SPLINE
SPL {X  -129.118, Y  +765.975, Z    +0.000, E1   +43.713, E3 -248326.138}
SPL {X  -146.252, Y  +736.362, Z    +0.000, E1   +34.795, E3 -248375.316}
SPL {X  -154.088, Y  +714.555, Z    +0.000, E1   +26.177, E3 -248389.332}
SPL {X  -156.688, Y  +703.837, Z    +0.000, E1   +21.096, E3 -248393.504}
SPL {X  -159.039, Y  +688.920, Z    +0.000, E1   +13.016, E3 -248397.436}
SPL {X  -159.888, Y  +677.224, Z    +0.000, E1    +5.773, E3 -248399.149}
SPL {X  -159.990, Y  +671.755, Z    +0.000, E1    +1.905, E3 -248399.552}
SPL {X  -159.990, Y  +669.598, Z    +0.000, E1    +0.205, E3 -248399.625}
SPL {X  -159.990, Y  +667.097, Z    +0.000, E1    -2.190, E3 -248399.720}
SPL {X  -159.990, Y  +662.904, Z    +0.000, E1    -7.618, E3 -248400.008}
SPL {X  -159.990, Y  +658.509, Z    +0.000, E1   -13.882, E3 -248400.544}
SPL {X  -159.990, Y  +652.317, Z    +0.000, E1   -22.778, E3 -248401.679}
SPL {X  -159.990, Y  +640.689, Z    +0.000, E1   -37.390, E3 -248403.222}
SPL {X  -159.990, Y  +585.634, Z    +0.000, E1   -68.681, E3 -248403.846}
SPL {X  -159.990, Y  +457.771, Z    +0.000, E1   -68.079, E3 -248494.407}
SPL {X  -159.990, Y  +453.218, Z    +0.000, E1   -67.322, E3 -248504.843}
SPL {X  -159.990, Y  +450.256, Z    +0.000, E1   -66.188, E3 -248516.775}
SPL {X  -159.990, Y  +445.667, Z    +0.000, E1   -65.356, E3 -248527.687}
SPL {X  -159.990, Y  +439.738, Z    +0.000, E1   -64.716, E3 -248538.500}
SPL {X  -159.990, Y  +435.528, Z    +0.000, E1   -63.972, E3 -248548.376}
SPL {X  -159.990, Y  +429.021, Z    +0.000, E1   -63.228, E3 -248560.989}
SPL {X  -159.990, Y  +423.267, Z    +0.000, E1   -62.365, E3 -248573.287}
SPL {X  -159.990, Y  +418.218, Z    +0.000, E1   -61.769, E3 -248583.299}
SPL {X  -159.990, Y  +412.274, Z    +0.000, E1   -61.123, E3 -248594.703}
SPL {X  -159.990, Y  +408.631, Z    +0.000, E1   -60.233, E3 -248605.165}
SPL {X  -159.990, Y  +404.834, Z    +0.000, E1   -59.529, E3 -248614.620}
SPL {X  -159.990, Y  +397.866, Z    +0.000, E1   -58.924, E3 -248627.708}
SPL {X  -159.990, Y  +387.403, Z    +0.000, E1   -58.805, E3 -248641.803}
SPL {X  -159.948, Y  +378.844, Z    +0.000, E1   -58.798, E3 -248652.843}
SPL {X  -159.570, Y  +370.916, Z    +0.000, E1   -58.738, E3 -248663.438}
SPL {X  -158.865, Y  +363.563, Z    +0.000, E1   -58.615, E3 -248673.648}
SPL {X  -157.976, Y  +357.197, Z    +0.000, E1   -58.476, E3 -248682.748}
SPL {X  -156.730, Y  +350.368, Z    +0.000, E1   -58.276, E3 -248692.844}
SPL {X  -155.026, Y  +342.956, Z    +0.000, E1   -58.003, E3 -248704.116}
SPL {X  -152.946, Y  +335.551, Z    +0.000, E1   -57.653, E3 -248715.764}
SPL {X  -150.899, Y  +329.336, Z    +0.000, E1   -57.290, E3 -248725.829}
SPL {X  -149.179, Y  +324.687, Z    +0.000, E1   -56.983, E3 -248733.519}
SPL {X  -147.281, Y  +320.009, Z    +0.000, E1   -56.662, E3 -248741.345}
SPL {X  -144.114, Y  +313.017, Z    +0.000, E1   -56.131, E3 -248753.312}
SPL {X  -140.858, Y  +306.633, Z    +0.000, E1   -55.477, E3 -248764.608}
SPL {X  -138.338, Y  +302.130, Z    +0.000, E1   -54.992, E3 -248772.657}
SPL {X  -124.427, Y  +281.929, Z    +0.000, E1   -46.852, E3 -248876.894}
ENDSPLINE

SPLINE
SPL {X  -148.251, Y  +322.346, Z    +0.000, E1   -33.039, E3 -248964.819}
SPL {X  -157.534, Y  +354.574, Z    +0.000, E1   -18.815, E3 -248981.648}
SPL {X  -159.548, Y  +370.614, Z    +0.000, E1    -9.656, E3 -248985.273}
SPL {X  -159.973, Y  +380.173, Z    +0.000, E1    -3.469, E3 -248986.340}
SPL {X  -159.990, Y  +384.791, Z    +0.000, E1    +0.055, E3 -248986.559}
SPL {X  -159.990, Y  +388.179, Z    +0.000, E1    +3.660, E3 -248986.719}
SPL {X  -159.990, Y  +394.222, Z    +0.000, E1   +11.674, E3 -248987.313}
SPL {X  -159.990, Y  +403.976, Z    +0.000, E1   +25.456, E3 -248989.192}
SPL {X  -159.990, Y  +417.120, Z    +0.000, E1   +39.678, E3 -248993.224}
SPL {X  -159.990, Y  +456.927, Z    +0.000, E1   +55.382, E3 -249015.084}
SPL {X  -159.990, Y  +530.047, Z    +0.000, E1   +58.901, E3 -249084.918}
SPL {X  -159.990, Y  +538.035, Z    +0.000, E1   +58.900, E3 -249095.143}
SPL {X  -159.990, Y  +546.883, Z    +0.000, E1   +58.912, E3 -249106.447}
SPL {X  -159.990, Y  +555.949, Z    +0.000, E1   +58.900, E3 -249118.066}
SPL {X  -159.990, Y  +563.718, Z    +0.000, E1   +58.903, E3 -249127.986}
SPL {X  -159.990, Y  +571.529, Z    +0.000, E1   +58.906, E3 -249137.970}
SPL {X  -159.990, Y  +579.859, Z    +0.000, E1   +58.907, E3 -249148.630}
SPL {X  -159.990, Y  +588.526, Z    +0.000, E1   +58.910, E3 -249159.703}
SPL {X  -159.990, Y  +596.521, Z    +0.000, E1   +58.902, E3 -249169.962}
SPL {X  -159.990, Y  +605.444, Z    +0.000, E1   +58.918, E3 -249181.352}
SPL {X  -159.990, Y  +613.908, Z    +0.000, E1   +58.900, E3 -249192.211}
SPL {X  -159.990, Y  +621.342, Z    +0.000, E1   +58.904, E3 -249201.719}
SPL {X  -159.990, Y  +629.920, Z    +0.000, E1   +58.912, E3 -249212.692}
SPL {X  -159.990, Y  +642.398, Z    +0.000, E1   +58.947, E3 -249228.599}
SPL {X  -159.990, Y  +654.206, Z    +0.000, E1   +58.908, E3 -249243.770}
SPL {X  -159.990, Y  +661.562, Z    +0.000, E1   +58.900, E3 -249253.199}
SPL {X  -159.990, Y  +670.328, Z    +0.000, E1   +58.911, E3 -249264.398}
SPL {X  -159.795, Y  +679.404, Z    +0.000, E1   +58.876, E3 -249276.223}
SPL {X  -159.282, Y  +686.534, Z    +0.000, E1   +58.787, E3 -249285.897}
SPL {X  -158.463, Y  +693.553, Z    +0.000, E1   +58.665, E3 -249295.738}
SPL {X  -157.294, Y  +700.745, Z    +0.000, E1   +58.469, E3 -249306.188}
SPL {X  -156.031, Y  +706.871, Z    +0.000, E1   +58.260, E3 -249315.334}
SPL {X  -154.558, Y  +712.835, Z    +0.000, E1   +58.028, E3 -249324.461}
SPL {X  -152.750, Y  +719.085, Z    +0.000, E1   +57.721, E3 -249334.307}
SPL {X  -150.741, Y  +725.111, Z    +0.000, E1   +57.387, E3 -249344.011}
SPL {X  -148.665, Y  +730.623, Z    +0.000, E1   +57.007, E3 -249353.160}
SPL {X  -146.664, Y  +735.425, Z    +0.000, E1   +56.657, E3 -249361.250}
SPL {X  -143.496, Y  +742.251, Z    +0.000, E1   +56.124, E3 -249372.943}
SPL {X  -140.752, Y  +747.564, Z    +0.000, E1   +55.554, E3 -249382.350}
SPL {X  -138.492, Y  +751.605, Z    +0.000, E1   +55.137, E3 -249389.541}
SPL {X  -124.324, Y  +772.199, Z    +0.000, E1   +48.708, E3 -249468.549}
ENDSPLINE

SPLINE
SPL {X  -129.118, Y  +765.975, Z    +0.000, E1   +43.713, E3 -249533.035}
SPL {X  -146.252, Y  +736.362, Z    +0.000, E1   +34.795, E3 -249582.213}
SPL {X  -155.916, Y  +707.374, Z    +0.000, E1   +22.878, E3 -249599.098}
SPL {X  -159.039, Y  +688.920, Z    +0.000, E1   +13.016, E3 -249604.333}
SPL {X  -159.888, Y  +677.224, Z    +0.000, E1    +5.773, E3 -249606.045}
SPL {X  -159.990, Y  +670.275, Z    +0.000, E1    +0.854, E3 -249606.499}
SPL {X  -159.990, Y  +667.097, Z    +0.000, E1    -2.190, E3 -249606.617}
SPL {X  -159.990, Y  +662.904, Z    +0.000, E1    -7.618, E3 -249606.905}
SPL {X  -159.990, Y  +658.509, Z    +0.000, E1   -13.882, E3 -249607.441}
SPL {X  -159.990, Y  +652.317, Z    +0.000, E1   -22.778, E3 -249608.576}
SPL {X  -159.990, Y  +640.689, Z    +0.000, E1   -37.390, E3 -249610.119}
SPL {X  -159.990, Y  +585.634, Z    +0.000, E1   -68.681, E3 -249610.743}
SPL {X  -159.990, Y  +457.771, Z    +0.000, E1   -68.079, E3 -249701.304}
SPL {X  -159.990, Y  +453.218, Z    +0.000, E1   -67.322, E3 -249711.739}
SPL {X  -159.990, Y  +450.256, Z    +0.000, E1   -66.188, E3 -249723.672}
SPL {X  -159.990, Y  +445.667, Z    +0.000, E1   -65.356, E3 -249734.584}
SPL {X  -159.990, Y  +439.738, Z    +0.000, E1   -64.716, E3 -249745.397}
SPL {X  -159.990, Y  +435.528, Z    +0.000, E1   -63.972, E3 -249755.272}
SPL {X  -159.990, Y  +429.021, Z    +0.000, E1   -63.228, E3 -249767.885}
SPL {X  -159.990, Y  +423.267, Z    +0.000, E1   -62.365, E3 -249780.183}
SPL {X  -159.990, Y  +418.218, Z    +0.000, E1   -61.769, E3 -249790.196}
SPL {X  -159.990, Y  +412.274, Z    +0.000, E1   -61.123, E3 -249801.600}
SPL {X  -159.990, Y  +408.631, Z    +0.000, E1   -60.233, E3 -249812.062}
SPL {X  -159.990, Y  +404.834, Z    +0.000, E1   -59.529, E3 -249821.517}
SPL {X  -159.990, Y  +397.866, Z    +0.000, E1   -58.924, E3 -249834.604}
SPL {X  -159.990, Y  +387.403, Z    +0.000, E1   -58.805, E3 -249848.700}
SPL {X  -159.948, Y  +378.844, Z    +0.000, E1   -58.798, E3 -249859.739}
SPL {X  -159.570, Y  +370.916, Z    +0.000, E1   -58.738, E3 -249870.335}
SPL {X  -158.865, Y  +363.563, Z    +0.000, E1   -58.615, E3 -249880.544}
SPL {X  -157.976, Y  +357.197, Z    +0.000, E1   -58.476, E3 -249889.645}
SPL {X  -156.730, Y  +350.368, Z    +0.000, E1   -58.276, E3 -249899.740}
SPL {X  -155.026, Y  +342.956, Z    +0.000, E1   -58.003, E3 -249911.012}
SPL {X  -152.946, Y  +335.551, Z    +0.000, E1   -57.653, E3 -249922.660}
SPL {X  -150.899, Y  +329.336, Z    +0.000, E1   -57.290, E3 -249932.726}
SPL {X  -149.179, Y  +324.687, Z    +0.000, E1   -56.983, E3 -249940.415}
SPL {X  -147.281, Y  +320.009, Z    +0.000, E1   -56.662, E3 -249948.241}
SPL {X  -144.114, Y  +313.017, Z    +0.000, E1   -56.131, E3 -249960.209}
SPL {X  -140.858, Y  +306.633, Z    +0.000, E1   -55.477, E3 -249971.504}
SPL {X  -138.338, Y  +302.130, Z    +0.000, E1   -54.992, E3 -249979.554}
SPL {X  -124.427, Y  +281.929, Z    +0.000, E1   -46.852, E3 -250083.790}
ENDSPLINE

SPLINE
SPL {X  -148.251, Y  +322.346, Z    +0.000, E1   -33.039, E3 -250171.715}
SPL {X  -156.481, Y  +349.177, Z    +0.000, E1   -21.514, E3 -250186.898}
SPL {X  -159.327, Y  +367.953, Z    +0.000, E1   -11.342, E3 -250191.690}
SPL {X  -159.973, Y  +380.173, Z    +0.000, E1    -3.469, E3 -250193.237}
SPL {X  -159.990, Y  +384.078, Z    +0.000, E1    -0.490, E3 -250193.434}
SPL {X  -159.990, Y  +386.348, Z    +0.000, E1    +1.571, E3 -250193.515}
SPL {X  -159.990, Y  +391.422, Z    +0.000, E1    +7.757, E3 -250193.889}
SPL {X  -159.990, Y  +399.099, Z    +0.000, E1   +18.787, E3 -250194.996}
SPL {X  -159.990, Y  +406.316, Z    +0.000, E1   +28.569, E3 -250196.673}
SPL {X  -159.990, Y  +417.120, Z    +0.000, E1   +39.678, E3 -250200.120}
SPL {X  -159.990, Y  +456.927, Z    +0.000, E1   +55.382, E3 -250221.980}
SPL {X  -159.990, Y  +530.047, Z    +0.000, E1   +58.901, E3 -250291.814}
SPL {X  -159.990, Y  +538.035, Z    +0.000, E1   +58.900, E3 -250302.040}
SPL {X  -159.990, Y  +546.883, Z    +0.000, E1   +58.912, E3 -250313.343}
SPL {X  -159.990, Y  +555.949, Z    +0.000, E1   +58.900, E3 -250324.963}
SPL {X  -159.990, Y  +563.718, Z    +0.000, E1   +58.903, E3 -250334.883}
SPL {X  -159.990, Y  +571.529, Z    +0.000, E1   +58.906, E3 -250344.867}
SPL {X  -159.990, Y  +579.859, Z    +0.000, E1   +58.907, E3 -250355.526}
SPL {X  -159.990, Y  +588.526, Z    +0.000, E1   +58.910, E3 -250366.600}
SPL {X  -159.990, Y  +596.521, Z    +0.000, E1   +58.902, E3 -250376.859}
SPL {X  -159.990, Y  +605.444, Z    +0.000, E1   +58.918, E3 -250388.248}
SPL {X  -159.990, Y  +613.908, Z    +0.000, E1   +58.900, E3 -250399.108}
SPL {X  -159.990, Y  +621.342, Z    +0.000, E1   +58.904, E3 -250408.616}
SPL {X  -159.990, Y  +629.920, Z    +0.000, E1   +58.912, E3 -250419.588}
SPL {X  -159.990, Y  +638.424, Z    +0.000, E1   +58.901, E3 -250430.488}
SPL {X  -159.990, Y  +645.995, Z    +0.000, E1   +58.900, E3 -250440.176}
SPL {X  -159.990, Y  +654.206, Z    +0.000, E1   +58.908, E3 -250450.667}
SPL {X  -159.990, Y  +661.562, Z    +0.000, E1   +58.900, E3 -250460.095}
SPL {X  -159.990, Y  +670.328, Z    +0.000, E1   +58.911, E3 -250471.294}
SPL {X  -159.795, Y  +679.404, Z    +0.000, E1   +58.876, E3 -250483.119}
SPL {X  -159.282, Y  +686.534, Z    +0.000, E1   +58.787, E3 -250492.793}
SPL {X  -158.463, Y  +693.553, Z    +0.000, E1   +58.665, E3 -250502.634}
SPL {X  -157.294, Y  +700.745, Z    +0.000, E1   +58.469, E3 -250513.084}
SPL {X  -156.031, Y  +706.871, Z    +0.000, E1   +58.260, E3 -250522.230}
SPL {X  -154.558, Y  +712.835, Z    +0.000, E1   +58.028, E3 -250531.357}
SPL {X  -152.750, Y  +719.085, Z    +0.000, E1   +57.721, E3 -250541.203}
SPL {X  -150.741, Y  +725.111, Z    +0.000, E1   +57.387, E3 -250550.907}
SPL {X  -148.665, Y  +730.623, Z    +0.000, E1   +57.007, E3 -250560.056}
SPL {X  -146.664, Y  +735.425, Z    +0.000, E1   +56.657, E3 -250568.146}
SPL {X  -143.496, Y  +742.251, Z    +0.000, E1   +56.124, E3 -250579.839}
SPL {X  -140.752, Y  +747.564, Z    +0.000, E1   +55.554, E3 -250589.247}
SPL {X  -138.492, Y  +751.605, Z    +0.000, E1   +55.137, E3 -250596.438}
SPL {X  -124.324, Y  +772.199, Z    +0.000, E1   +48.708, E3 -250675.446}
ENDSPLINE

SPLINE
SPL {X  -129.118, Y  +765.975, Z    +0.000, E1   +43.713, E3 -250739.931}
SPL {X  -146.252, Y  +736.362, Z    +0.000, E1   +34.795, E3 -250789.109}
SPL {X  -154.088, Y  +714.555, Z    +0.000, E1   +26.177, E3 -250803.125}
SPL {X  -156.688, Y  +703.837, Z    +0.000, E1   +21.096, E3 -250807.297}
SPL {X  -159.039, Y  +688.920, Z    +0.000, E1   +13.016, E3 -250811.229}
SPL {X  -159.888, Y  +677.224, Z    +0.000, E1    +5.773, E3 -250812.942}
SPL {X  -159.990, Y  +671.755, Z    +0.000, E1    +1.905, E3 -250813.345}
SPL {X  -159.990, Y  +668.898, Z    +0.000, E1    -0.346, E3 -250813.439}
SPL {X  -159.990, Y  +666.084, Z    +0.000, E1    -3.512, E3 -250813.562}
SPL {X  -159.990, Y  +662.904, Z    +0.000, E1    -7.618, E3 -250813.801}
SPL {X  -159.990, Y  +658.509, Z    +0.000, E1   -13.882, E3 -250814.337}
SPL {X  -159.990, Y  +652.317, Z    +0.000, E1   -22.778, E3 -250815.473}
SPL {X  -159.990, Y  +640.689, Z    +0.000, E1   -37.390, E3 -250817.015}
SPL {X  -159.990, Y  +585.634, Z    +0.000, E1   -68.681, E3 -250817.639}
SPL {X  -159.990, Y  +457.771, Z    +0.000, E1   -68.079, E3 -250908.201}
SPL {X  -159.990, Y  +453.218, Z    +0.000, E1   -67.322, E3 -250918.636}
SPL {X  -159.990, Y  +450.256, Z    +0.000, E1   -66.188, E3 -250930.569}
SPL {X  -159.990, Y  +445.667, Z    +0.000, E1   -65.356, E3 -250941.480}
SPL {X  -159.990, Y  +439.738, Z    +0.000, E1   -64.716, E3 -250952.293}
SPL {X  -159.990, Y  +435.528, Z    +0.000, E1   -63.972, E3 -250962.169}
SPL {X  -159.990, Y  +429.021, Z    +0.000, E1   -63.228, E3 -250974.782}
SPL {X  -159.990, Y  +423.267, Z    +0.000, E1   -62.365, E3 -250987.080}
SPL {X  -159.990, Y  +418.218, Z    +0.000, E1   -61.769, E3 -250997.092}
SPL {X  -159.990, Y  +412.274, Z    +0.000, E1   -61.123, E3 -251008.496}
SPL {X  -159.990, Y  +408.631, Z    +0.000, E1   -60.233, E3 -251018.958}
SPL {X  -159.990, Y  +402.821, Z    +0.000, E1   -59.334, E3 -251032.486}
SPL {X  -159.990, Y  +395.849, Z    +0.000, E1   -58.799, E3 -251044.750}
SPL {X  -159.990, Y  +387.403, Z    +0.000, E1   -58.805, E3 -251055.596}
SPL {X  -159.948, Y  +378.844, Z    +0.000, E1   -58.798, E3 -251066.636}
SPL {X  -159.570, Y  +370.916, Z    +0.000, E1   -58.738, E3 -251077.231}
SPL {X  -158.865, Y  +363.563, Z    +0.000, E1   -58.615, E3 -251087.441}
SPL {X  -157.976, Y  +357.197, Z    +0.000, E1   -58.476, E3 -251096.542}
SPL {X  -156.730, Y  +350.368, Z    +0.000, E1   -58.276, E3 -251106.637}
SPL {X  -155.026, Y  +342.956, Z    +0.000, E1   -58.003, E3 -251117.909}
SPL {X  -152.946, Y  +335.551, Z    +0.000, E1   -57.653, E3 -251129.557}
SPL {X  -150.105, Y  +327.135, Z    +0.000, E1   -57.196, E3 -251143.177}
SPL {X  -147.281, Y  +320.009, Z    +0.000, E1   -56.662, E3 -251155.138}
SPL {X  -144.114, Y  +313.017, Z    +0.000, E1   -56.131, E3 -251167.105}
SPL {X  -140.858, Y  +306.633, Z    +0.000, E1   -55.477, E3 -251178.401}
SPL {X  -138.338, Y  +302.130, Z    +0.000, E1   -54.992, E3 -251186.450}
SPL {X  -124.427, Y  +281.929, Z    +0.000, E1   -46.852, E3 -251290.687}
ENDSPLINE

SPLINE
SPL {X  -148.251, Y  +322.346, Z    +0.000, E1   -33.039, E3 -251378.612}
SPL {X  -156.481, Y  +349.177, Z    +0.000, E1   -21.514, E3 -251393.795}
SPL {X  -159.327, Y  +367.953, Z    +0.000, E1   -11.342, E3 -251398.586}
SPL {X  -159.973, Y  +380.173, Z    +0.000, E1    -3.469, E3 -251400.133}
SPL {X  -159.990, Y  +384.078, Z    +0.000, E1    -0.490, E3 -251400.331}
SPL {X  -159.990, Y  +385.440, Z    +0.000, E1    +0.747, E3 -251400.372}
SPL {X  -159.990, Y  +388.179, Z    +0.000, E1    +3.660, E3 -251400.512}
SPL {X  -159.990, Y  +394.222, Z    +0.000, E1   +11.674, E3 -251401.106}
SPL {X  -159.990, Y  +403.976, Z    +0.000, E1   +25.456, E3 -251402.985}
SPL {X  -159.990, Y  +417.120, Z    +0.000, E1   +39.678, E3 -251407.017}
SPL {X  -159.990, Y  +456.927, Z    +0.000, E1   +55.382, E3 -251428.877}
SPL {X  -159.990, Y  +530.047, Z    +0.000, E1   +58.901, E3 -251498.711}
SPL {X  -159.990, Y  +538.035, Z    +0.000, E1   +58.900, E3 -251508.936}
SPL {X  -159.990, Y  +546.883, Z    +0.000, E1   +58.912, E3 -251520.240}
SPL {X  -159.990, Y  +555.949, Z    +0.000, E1   +58.900, E3 -251531.859}
SPL {X  -159.990, Y  +563.718, Z    +0.000, E1   +58.903, E3 -251541.779}
SPL {X  -159.990, Y  +571.529, Z    +0.000, E1   +58.906, E3 -251551.764}
SPL {X  -159.990, Y  +579.859, Z    +0.000, E1   +58.907, E3 -251562.423}
SPL {X  -159.990, Y  +588.526, Z    +0.000, E1   +58.910, E3 -251573.496}
SPL {X  -159.990, Y  +596.521, Z    +0.000, E1   +58.902, E3 -251583.755}
SPL {X  -159.990, Y  +605.444, Z    +0.000, E1   +58.918, E3 -251595.145}
SPL {X  -159.990, Y  +618.101, Z    +0.000, E1   +58.946, E3 -251611.292}
SPL {X  -159.990, Y  +629.920, Z    +0.000, E1   +58.912, E3 -251626.485}
SPL {X  -159.990, Y  +638.424, Z    +0.000, E1   +58.901, E3 -251637.385}
SPL {X  -159.990, Y  +645.995, Z    +0.000, E1   +58.900, E3 -251647.073}
SPL {X  -159.990, Y  +654.206, Z    +0.000, E1   +58.908, E3 -251657.563}
SPL {X  -159.990, Y  +661.562, Z    +0.000, E1   +58.900, E3 -251666.992}
SPL {X  -159.990, Y  +670.328, Z    +0.000, E1   +58.911, E3 -251678.191}
SPL {X  -159.795, Y  +679.404, Z    +0.000, E1   +58.876, E3 -251690.016}
SPL {X  -159.282, Y  +686.534, Z    +0.000, E1   +58.787, E3 -251699.690}
SPL {X  -158.463, Y  +693.553, Z    +0.000, E1   +58.665, E3 -251709.531}
SPL {X  -157.294, Y  +700.745, Z    +0.000, E1   +58.469, E3 -251719.981}
SPL {X  -156.031, Y  +706.871, Z    +0.000, E1   +58.260, E3 -251729.127}
SPL {X  -154.558, Y  +712.835, Z    +0.000, E1   +58.028, E3 -251738.254}
SPL {X  -152.750, Y  +719.085, Z    +0.000, E1   +57.721, E3 -251748.100}
SPL {X  -150.741, Y  +725.111, Z    +0.000, E1   +57.387, E3 -251757.804}
SPL {X  -148.665, Y  +730.623, Z    +0.000, E1   +57.007, E3 -251766.953}
SPL {X  -146.664, Y  +735.425, Z    +0.000, E1   +56.657, E3 -251775.043}
SPL {X  -143.496, Y  +742.251, Z    +0.000, E1   +56.124, E3 -251786.736}
SPL {X  -140.752, Y  +747.564, Z    +0.000, E1   +55.554, E3 -251796.143}
SPL {X  -138.492, Y  +751.605, Z    +0.000, E1   +55.137, E3 -251803.334}
SPL {X  -124.324, Y  +772.199, Z    +0.000, E1   +48.708, E3 -251882.343}
ENDSPLINE

SPLINE
SPL {X  -129.118, Y  +765.975, Z    +0.000, E1   +43.713, E3 -251946.828}
SPL {X  -146.252, Y  +736.362, Z    +0.000, E1   +34.795, E3 -251996.006}
SPL {X  -155.916, Y  +707.374, Z    +0.000, E1   +22.878, E3 -252012.891}
SPL {X  -159.039, Y  +688.920, Z    +0.000, E1   +13.016, E3 -252018.126}
SPL {X  -159.888, Y  +677.224, Z    +0.000, E1    +5.773, E3 -252019.839}
SPL {X  -159.990, Y  +670.275, Z    +0.000, E1    +0.854, E3 -252020.292}
SPL {X  -159.990, Y  +667.097, Z    +0.000, E1    -2.190, E3 -252020.410}
SPL {X  -159.990, Y  +662.904, Z    +0.000, E1    -7.618, E3 -252020.698}
SPL {X  -159.990, Y  +658.509, Z    +0.000, E1   -13.882, E3 -252021.234}
SPL {X  -159.990, Y  +652.317, Z    +0.000, E1   -22.778, E3 -252022.369}
SPL {X  -159.990, Y  +640.689, Z    +0.000, E1   -37.390, E3 -252023.912}
SPL {X  -159.990, Y  +585.634, Z    +0.000, E1   -68.681, E3 -252024.536}
SPL {X  -159.990, Y  +457.771, Z    +0.000, E1   -68.079, E3 -252115.097}
SPL {X  -159.990, Y  +453.218, Z    +0.000, E1   -67.322, E3 -252125.532}
SPL {X  -159.990, Y  +450.256, Z    +0.000, E1   -66.188, E3 -252137.465}
SPL {X  -159.990, Y  +445.667, Z    +0.000, E1   -65.356, E3 -252148.377}
SPL {X  -159.990, Y  +439.738, Z    +0.000, E1   -64.716, E3 -252159.190}
SPL {X  -159.990, Y  +435.528, Z    +0.000, E1   -63.972, E3 -252169.065}
SPL {X  -159.990, Y  +429.021, Z    +0.000, E1   -63.228, E3 -252181.678}
SPL {X  -159.990, Y  +423.267, Z    +0.000, E1   -62.365, E3 -252193.976}
SPL {X  -159.990, Y  +418.218, Z    +0.000, E1   -61.769, E3 -252203.989}
SPL {X  -159.990, Y  +412.274, Z    +0.000, E1   -61.123, E3 -252215.393}
SPL {X  -159.990, Y  +408.631, Z    +0.000, E1   -60.233, E3 -252225.855}
SPL {X  -159.990, Y  +404.834, Z    +0.000, E1   -59.529, E3 -252235.310}
SPL {X  -159.990, Y  +397.866, Z    +0.000, E1   -58.924, E3 -252248.397}
SPL {X  -159.990, Y  +387.403, Z    +0.000, E1   -58.805, E3 -252262.493}
SPL {X  -159.948, Y  +378.844, Z    +0.000, E1   -58.798, E3 -252273.532}
SPL {X  -159.570, Y  +370.916, Z    +0.000, E1   -58.738, E3 -252284.128}
SPL {X  -158.865, Y  +363.563, Z    +0.000, E1   -58.615, E3 -252294.337}
SPL {X  -157.976, Y  +357.197, Z    +0.000, E1   -58.476, E3 -252303.438}
SPL {X  -156.730, Y  +350.368, Z    +0.000, E1   -58.276, E3 -252313.533}
SPL {X  -155.026, Y  +342.956, Z    +0.000, E1   -58.003, E3 -252324.806}
SPL {X  -152.946, Y  +335.551, Z    +0.000, E1   -57.653, E3 -252336.453}
SPL {X  -150.105, Y  +327.135, Z    +0.000, E1   -57.196, E3 -252350.074}
SPL {X  -146.578, Y  +318.377, Z    +0.000, E1   -56.572, E3 -252364.767}
SPL {X  -143.463, Y  +311.683, Z    +0.000, E1   -55.972, E3 -252376.380}
SPL {X  -140.858, Y  +306.633, Z    +0.000, E1   -55.477, E3 -252385.297}
SPL {X  -138.338, Y  +302.130, Z    +0.000, E1   -54.992, E3 -252393.347}
SPL {X  -124.427, Y  +281.929, Z    +0.000, E1   -46.852, E3 -252497.583}
ENDSPLINE

SPLINE
SPL {X  -138.506, Y  +302.419, Z    +0.000, E1   -39.451, E3 -252563.558}
SPL {X  -149.686, Y  +326.013, Z    +0.000, E1   -31.658, E3 -252588.694}
SPL {X  -157.534, Y  +354.574, Z    +0.000, E1   -18.815, E3 -252602.337}
SPL {X  -159.548, Y  +370.614, Z    +0.000, E1    -9.656, E3 -252605.963}
SPL {X  -159.928, Y  +378.035, Z    +0.000, E1    -4.866, E3 -252606.878}
SPL {X  -159.990, Y  +383.381, Z    +0.000, E1    -1.123, E3 -252607.199}
SPL {X  -159.990, Y  +386.348, Z    +0.000, E1    +1.571, E3 -252607.308}
SPL {X  -159.990, Y  +389.406, Z    +0.000, E1    +5.320, E3 -252607.488}
SPL {X  -159.990, Y  +394.222, Z    +0.000, E1   +11.674, E3 -252608.002}
SPL {X  -159.990, Y  +403.976, Z    +0.000, E1   +25.456, E3 -252609.882}
SPL {X  -159.990, Y  +417.120, Z    +0.000, E1   +39.678, E3 -252613.913}
SPL {X  -159.990, Y  +456.927, Z    +0.000, E1   +55.382, E3 -252635.773}
SPL {X  -159.990, Y  +530.047, Z    +0.000, E1   +58.901, E3 -252705.607}
SPL {X  -159.990, Y  +538.035, Z    +0.000, E1   +58.900, E3 -252715.833}
SPL {X  -159.990, Y  +546.883, Z    +0.000, E1   +58.912, E3 -252727.136}
SPL {X  -159.990, Y  +555.949, Z    +0.000, E1   +58.900, E3 -252738.756}
SPL {X  -159.990, Y  +563.718, Z    +0.000, E1   +58.903, E3 -252748.676}
SPL {X  -159.990, Y  +571.529, Z    +0.000, E1   +58.906, E3 -252758.660}
SPL {X  -159.990, Y  +579.859, Z    +0.000, E1   +58.907, E3 -252769.319}
SPL {X  -159.990, Y  +588.526, Z    +0.000, E1   +58.910, E3 -252780.393}
SPL {X  -159.990, Y  +596.521, Z    +0.000, E1   +58.902, E3 -252790.652}
SPL {X  -159.990, Y  +605.444, Z    +0.000, E1   +58.918, E3 -252802.042}
SPL {X  -159.990, Y  +618.101, Z    +0.000, E1   +58.946, E3 -252818.188}
SPL {X  -159.990, Y  +629.920, Z    +0.000, E1   +58.912, E3 -252833.381}
SPL {X  -159.990, Y  +638.424, Z    +0.000, E1   +58.901, E3 -252844.281}
SPL {X  -159.990, Y  +645.995, Z    +0.000, E1   +58.900, E3 -252853.969}
SPL {X  -159.990, Y  +654.206, Z    +0.000, E1   +58.908, E3 -252864.460}
SPL {X  -159.990, Y  +661.562, Z    +0.000, E1   +58.900, E3 -252873.888}
SPL {X  -159.990, Y  +670.328, Z    +0.000, E1   +58.911, E3 -252885.087}
SPL {X  -159.795, Y  +679.404, Z    +0.000, E1   +58.876, E3 -252896.913}
SPL {X  -159.282, Y  +686.534, Z    +0.000, E1   +58.787, E3 -252906.586}
SPL {X  -158.463, Y  +693.553, Z    +0.000, E1   +58.665, E3 -252916.427}
SPL {X  -157.294, Y  +700.745, Z    +0.000, E1   +58.469, E3 -252926.877}
SPL {X  -156.031, Y  +706.871, Z    +0.000, E1   +58.260, E3 -252936.023}
SPL {X  -154.558, Y  +712.835, Z    +0.000, E1   +58.028, E3 -252945.150}
SPL {X  -152.750, Y  +719.085, Z    +0.000, E1   +57.721, E3 -252954.996}
SPL {X  -150.741, Y  +725.111, Z    +0.000, E1   +57.387, E3 -252964.701}
SPL {X  -148.665, Y  +730.623, Z    +0.000, E1   +57.007, E3 -252973.849}
SPL {X  -146.664, Y  +735.425, Z    +0.000, E1   +56.657, E3 -252981.939}
SPL {X  -144.631, Y  +739.900, Z    +0.000, E1   +56.280, E3 -252989.625}
SPL {X  -141.795, Y  +745.600, Z    +0.000, E1   +55.801, E3 -252999.508}
SPL {X  -138.492, Y  +751.605, Z    +0.000, E1   +55.137, E3 -253010.231}
SPL {X  -124.324, Y  +772.199, Z    +0.000, E1   +48.708, E3 -253089.239}
ENDSPLINE

SPLINE
SPL {X  -129.118, Y  +765.975, Z    +0.000, E1   +43.713, E3 -253153.724}
SPL {X  -146.252, Y  +736.362, Z    +0.000, E1   +34.795, E3 -253202.902}
SPL {X  -154.088, Y  +714.555, Z    +0.000, E1   +26.177, E3 -253216.918}
SPL {X  -156.688, Y  +703.837, Z    +0.000, E1   +21.096, E3 -253221.090}
SPL {X  -159.039, Y  +688.920, Z    +0.000, E1   +13.016, E3 -253225.022}
SPL {X  -159.888, Y  +677.224, Z    +0.000, E1    +5.773, E3 -253226.735}
SPL {X  -159.990, Y  +671.755, Z    +0.000, E1    +1.905, E3 -253227.138}
SPL {X  -159.990, Y  +668.898, Z    +0.000, E1    -0.346, E3 -253227.233}
SPL {X  -159.990, Y  +666.084, Z    +0.000, E1    -3.512, E3 -253227.355}
SPL {X  -159.990, Y  +662.904, Z    +0.000, E1    -7.618, E3 -253227.594}
SPL {X  -159.990, Y  +658.509, Z    +0.000, E1   -13.882, E3 -253228.130}
SPL {X  -159.990, Y  +652.317, Z    +0.000, E1   -22.778, E3 -253229.266}
SPL {X  -159.990, Y  +640.689, Z    +0.000, E1   -37.390, E3 -253230.808}
SPL {X  -159.990, Y  +585.634, Z    +0.000, E1   -68.681, E3 -253231.432}
SPL {X  -159.990, Y  +457.771, Z    +0.000, E1   -68.079, E3 -253321.994}
SPL {X  -159.990, Y  +453.218, Z    +0.000, E1   -67.322, E3 -253332.429}
SPL {X  -159.990, Y  +450.256, Z    +0.000, E1   -66.188, E3 -253344.362}
SPL {X  -159.990, Y  +445.667, Z    +0.000, E1   -65.356, E3 -253355.273}
SPL {X  -159.990, Y  +439.738, Z    +0.000, E1   -64.716, E3 -253366.086}
SPL {X  -159.990, Y  +435.528, Z    +0.000, E1   -63.972, E3 -253375.962}
SPL {X  -159.990, Y  +429.021, Z    +0.000, E1   -63.228, E3 -253388.575}
SPL {X  -159.990, Y  +423.267, Z    +0.000, E1   -62.365, E3 -253400.873}
SPL {X  -159.990, Y  +418.218, Z    +0.000, E1   -61.769, E3 -253410.885}
SPL {X  -159.990, Y  +412.274, Z    +0.000, E1   -61.123, E3 -253422.289}
SPL {X  -159.990, Y  +408.631, Z    +0.000, E1   -60.233, E3 -253432.752}
SPL {X  -159.990, Y  +404.834, Z    +0.000, E1   -59.529, E3 -253442.207}
SPL {X  -159.990, Y  +397.866, Z    +0.000, E1   -58.924, E3 -253455.294}
SPL {X  -159.990, Y  +387.403, Z    +0.000, E1   -58.805, E3 -253469.389}
SPL {X  -159.948, Y  +378.844, Z    +0.000, E1   -58.798, E3 -253480.429}
SPL {X  -159.570, Y  +370.916, Z    +0.000, E1   -58.738, E3 -253491.024}
SPL {X  -158.865, Y  +363.563, Z    +0.000, E1   -58.615, E3 -253501.234}
SPL {X  -157.976, Y  +357.197, Z    +0.000, E1   -58.476, E3 -253510.335}
SPL {X  -156.730, Y  +350.368, Z    +0.000, E1   -58.276, E3 -253520.430}
SPL {X  -155.026, Y  +342.956, Z    +0.000, E1   -58.003, E3 -253531.702}
SPL {X  -152.946, Y  +335.551, Z    +0.000, E1   -57.653, E3 -253543.350}
SPL {X  -150.899, Y  +329.336, Z    +0.000, E1   -57.290, E3 -253553.416}
SPL {X  -149.179, Y  +324.687, Z    +0.000, E1   -56.983, E3 -253561.105}
SPL {X  -147.281, Y  +320.009, Z    +0.000, E1   -56.662, E3 -253568.931}
SPL {X  -144.114, Y  +313.017, Z    +0.000, E1   -56.131, E3 -253580.898}
SPL {X  -140.858, Y  +306.633, Z    +0.000, E1   -55.477, E3 -253592.194}
SPL {X  -138.338, Y  +302.130, Z    +0.000, E1   -54.992, E3 -253600.243}
SPL {X  -124.427, Y  +281.929, Z    +0.000, E1   -46.852, E3 -253704.480}
ENDSPLINE

SPLINE
SPL {X  -148.251, Y  +322.346, Z    +0.000, E1   -33.039, E3 -253792.405}
SPL {X  -157.534, Y  +354.574, Z    +0.000, E1   -18.815, E3 -253809.234}
SPL {X  -159.548, Y  +370.614, Z    +0.000, E1    -9.656, E3 -253812.859}
SPL {X  -159.928, Y  +378.035, Z    +0.000, E1    -4.866, E3 -253813.775}
SPL {X  -159.990, Y  +383.381, Z    +0.000, E1    -1.123, E3 -253814.096}
SPL {X  -159.990, Y  +385.440, Z    +0.000, E1    +0.747, E3 -253814.165}
SPL {X  -159.990, Y  +388.179, Z    +0.000, E1    +3.660, E3 -253814.305}
SPL {X  -159.990, Y  +394.222, Z    +0.000, E1   +11.674, E3 -253814.899}
SPL {X  -159.990, Y  +403.976, Z    +0.000, E1   +25.456, E3 -253816.778}
SPL {X  -159.990, Y  +417.120, Z    +0.000, E1   +39.678, E3 -253820.810}
SPL {X  -159.990, Y  +456.927, Z    +0.000, E1   +55.382, E3 -253842.670}
SPL {X  -159.990, Y  +530.047, Z    +0.000, E1   +58.901, E3 -253912.504}
SPL {X  -159.990, Y  +538.035, Z    +0.000, E1   +58.900, E3 -253922.729}
SPL {X  -159.990, Y  +546.883, Z    +0.000, E1   +58.912, E3 -253934.033}
SPL {X  -159.990, Y  +555.949, Z    +0.000, E1   +58.900, E3 -253945.652}
SPL {X  -159.990, Y  +563.718, Z    +0.000, E1   +58.903, E3 -253955.573}
SPL {X  -159.990, Y  +571.529, Z    +0.000, E1   +58.906, E3 -253965.557}
SPL {X  -159.990, Y  +579.859, Z    +0.000, E1   +58.907, E3 -253976.216}
SPL {X  -159.990, Y  +588.526, Z    +0.000, E1   +58.910, E3 -253987.290}
SPL {X  -159.990, Y  +596.521, Z    +0.000, E1   +58.902, E3 -253997.549}
SPL {X  -159.990, Y  +605.444, Z    +0.000, E1   +58.918, E3 -254008.938}
SPL {X  -159.990, Y  +613.908, Z    +0.000, E1   +58.900, E3 -254019.797}
SPL {X  -159.990, Y  +621.342, Z    +0.000, E1   +58.904, E3 -254029.305}
SPL {X  -159.990, Y  +629.920, Z    +0.000, E1   +58.912, E3 -254040.278}
SPL {X  -159.990, Y  +642.398, Z    +0.000, E1   +58.947, E3 -254056.185}
SPL {X  -159.990, Y  +654.206, Z    +0.000, E1   +58.908, E3 -254071.356}
SPL {X  -159.990, Y  +661.562, Z    +0.000, E1   +58.900, E3 -254080.785}
SPL {X  -159.990, Y  +670.328, Z    +0.000, E1   +58.911, E3 -254091.984}
SPL {X  -159.795, Y  +679.404, Z    +0.000, E1   +58.876, E3 -254103.809}
SPL {X  -159.282, Y  +686.534, Z    +0.000, E1   +58.787, E3 -254113.483}
SPL {X  -158.463, Y  +693.553, Z    +0.000, E1   +58.665, E3 -254123.324}
SPL {X  -157.294, Y  +700.745, Z    +0.000, E1   +58.469, E3 -254133.774}
SPL {X  -156.031, Y  +706.871, Z    +0.000, E1   +58.260, E3 -254142.920}
SPL {X  -154.558, Y  +712.835, Z    +0.000, E1   +58.028, E3 -254152.047}
SPL {X  -152.750, Y  +719.085, Z    +0.000, E1   +57.721, E3 -254161.893}
SPL {X  -150.741, Y  +725.111, Z    +0.000, E1   +57.387, E3 -254171.597}
SPL {X  -148.665, Y  +730.623, Z    +0.000, E1   +57.007, E3 -254180.746}
SPL {X  -146.664, Y  +735.425, Z    +0.000, E1   +56.657, E3 -254188.836}
SPL {X  -144.631, Y  +739.900, Z    +0.000, E1   +56.280, E3 -254196.521}
SPL {X  -141.795, Y  +745.600, Z    +0.000, E1   +55.801, E3 -254206.404}
SPL {X  -138.492, Y  +751.605, Z    +0.000, E1   +55.137, E3 -254217.128}
SPL {X  -124.324, Y  +772.199, Z    +0.000, E1   +48.708, E3 -254296.136}
ENDSPLINE

SPLINE
SPL {X  -129.118, Y  +765.975, Z    +0.000, E1   +43.713, E3 -254360.621}
SPL {X  -146.252, Y  +736.362, Z    +0.000, E1   +34.795, E3 -254409.799}
SPL {X  -154.088, Y  +714.555, Z    +0.000, E1   +26.177, E3 -254423.815}
SPL {X  -156.688, Y  +703.837, Z    +0.000, E1   +21.096, E3 -254427.987}
SPL {X  -159.039, Y  +688.920, Z    +0.000, E1   +13.016, E3 -254431.919}
SPL {X  -159.888, Y  +677.224, Z    +0.000, E1    +5.773, E3 -254433.632}
SPL {X  -159.990, Y  +670.275, Z    +0.000, E1    +0.854, E3 -254434.085}
SPL {X  -159.990, Y  +667.097, Z    +0.000, E1    -2.190, E3 -254434.203}
SPL {X  -159.990, Y  +662.904, Z    +0.000, E1    -7.618, E3 -254434.491}
SPL {X  -159.990, Y  +658.509, Z    +0.000, E1   -13.882, E3 -254435.027}
SPL {X  -159.990, Y  +652.317, Z    +0.000, E1   -22.778, E3 -254436.162}
SPL {X  -159.990, Y  +640.689, Z    +0.000, E1   -37.390, E3 -254437.705}
SPL {X  -159.990, Y  +585.634, Z    +0.000, E1   -68.681, E3 -254438.329}
SPL {X  -159.990, Y  +457.771, Z    +0.000, E1   -68.079, E3 -254528.890}
SPL {X  -159.990, Y  +453.218, Z    +0.000, E1   -67.322, E3 -254539.326}
SPL {X  -159.990, Y  +450.256, Z    +0.000, E1   -66.188, E3 -254551.258}
SPL {X  -159.990, Y  +445.667, Z    +0.000, E1   -65.356, E3 -254562.170}
SPL {X  -159.990, Y  +439.738, Z    +0.000, E1   -64.716, E3 -254572.983}
SPL {X  -159.990, Y  +433.217, Z    +0.000, E1   -63.756, E3 -254587.127}
SPL {X  -159.990, Y  +425.111, Z    +0.000, E1   -62.687, E3 -254603.668}
SPL {X  -159.990, Y  +418.218, Z    +0.000, E1   -61.769, E3 -254617.782}
SPL {X  -159.990, Y  +412.274, Z    +0.000, E1   -61.123, E3 -254629.186}
SPL {X  -159.990, Y  +408.631, Z    +0.000, E1   -60.233, E3 -254639.648}
SPL {X  -159.990, Y  +402.821, Z    +0.000, E1   -59.334, E3 -254653.175}
SPL {X  -159.990, Y  +395.849, Z    +0.000, E1   -58.799, E3 -254665.440}
SPL {X  -159.990, Y  +387.403, Z    +0.000, E1   -58.805, E3 -254676.286}
SPL {X  -159.948, Y  +378.844, Z    +0.000, E1   -58.798, E3 -254687.326}
SPL {X  -159.570, Y  +370.916, Z    +0.000, E1   -58.738, E3 -254697.921}
SPL {X  -158.865, Y  +363.563, Z    +0.000, E1   -58.615, E3 -254708.130}
SPL {X  -157.976, Y  +357.197, Z    +0.000, E1   -58.476, E3 -254717.231}
SPL {X  -156.730, Y  +350.368, Z    +0.000, E1   -58.276, E3 -254727.326}
SPL {X  -155.026, Y  +342.956, Z    +0.000, E1   -58.003, E3 -254738.599}
SPL {X  -152.946, Y  +335.551, Z    +0.000, E1   -57.653, E3 -254750.247}
SPL {X  -150.105, Y  +327.135, Z    +0.000, E1   -57.196, E3 -254763.867}
SPL {X  -146.578, Y  +318.377, Z    +0.000, E1   -56.572, E3 -254778.560}
SPL {X  -143.463, Y  +311.683, Z    +0.000, E1   -55.972, E3 -254790.173}
SPL {X  -140.858, Y  +306.633, Z    +0.000, E1   -55.477, E3 -254799.091}
SPL {X  -138.338, Y  +302.130, Z    +0.000, E1   -54.992, E3 -254807.140}
SPL {X  -124.427, Y  +281.929, Z    +0.000, E1   -46.852, E3 -254911.376}
ENDSPLINE

SPLINE
SPL {X  -148.251, Y  +322.346, Z    +0.000, E1   -33.039, E3 -254999.301}
SPL {X  -157.534, Y  +354.574, Z    +0.000, E1   -18.815, E3 -255016.130}
SPL {X  -159.548, Y  +370.614, Z    +0.000, E1    -9.656, E3 -255019.756}
SPL {X  -159.928, Y  +378.035, Z    +0.000, E1    -4.866, E3 -255020.671}
SPL {X  -159.990, Y  +383.381, Z    +0.000, E1    -1.123, E3 -255020.992}
SPL {X  -159.990, Y  +385.440, Z    +0.000, E1    +0.747, E3 -255021.061}
SPL {X  -159.990, Y  +388.179, Z    +0.000, E1    +3.660, E3 -255021.202}
SPL {X  -159.990, Y  +394.222, Z    +0.000, E1   +11.674, E3 -255021.795}
SPL {X  -159.990, Y  +403.976, Z    +0.000, E1   +25.456, E3 -255023.675}
SPL {X  -159.990, Y  +417.120, Z    +0.000, E1   +39.678, E3 -255027.706}
SPL {X  -159.990, Y  +456.927, Z    +0.000, E1   +55.382, E3 -255049.567}
SPL {X  -159.990, Y  +530.047, Z    +0.000, E1   +58.901, E3 -255119.400}
SPL {X  -159.990, Y  +538.035, Z    +0.000, E1   +58.900, E3 -255129.626}
SPL {X  -159.990, Y  +546.883, Z    +0.000, E1   +58.912, E3 -255140.929}
SPL {X  -159.990, Y  +555.949, Z    +0.000, E1   +58.900, E3 -255152.549}
SPL {X  -159.990, Y  +563.718, Z    +0.000, E1   +58.903, E3 -255162.469}
SPL {X  -159.990, Y  +571.529, Z    +0.000, E1   +58.906, E3 -255172.453}
SPL {X  -159.990, Y  +579.859, Z    +0.000, E1   +58.907, E3 -255183.112}
SPL {X  -159.990, Y  +588.526, Z    +0.000, E1   +58.910, E3 -255194.186}
SPL {X  -159.990, Y  +596.521, Z    +0.000, E1   +58.902, E3 -255204.445}
SPL {X  -159.990, Y  +605.444, Z    +0.000, E1   +58.918, E3 -255215.835}
SPL {X  -159.990, Y  +613.908, Z    +0.000, E1   +58.900, E3 -255226.694}
SPL {X  -159.990, Y  +621.342, Z    +0.000, E1   +58.904, E3 -255236.202}
SPL {X  -159.990, Y  +629.920, Z    +0.000, E1   +58.912, E3 -255247.174}
SPL {X  -159.990, Y  +642.398, Z    +0.000, E1   +58.947, E3 -255263.082}
SPL {X  -159.990, Y  +654.206, Z    +0.000, E1   +58.908, E3 -255278.253}
SPL {X  -159.990, Y  +661.562, Z    +0.000, E1   +58.900, E3 -255287.681}
SPL {X  -159.990, Y  +670.328, Z    +0.000, E1   +58.911, E3 -255298.880}
SPL {X  -159.795, Y  +679.404, Z    +0.000, E1   +58.876, E3 -255310.706}
SPL {X  -159.282, Y  +686.534, Z    +0.000, E1   +58.787, E3 -255320.379}
SPL {X  -158.463, Y  +693.553, Z    +0.000, E1   +58.665, E3 -255330.221}
SPL {X  -157.294, Y  +700.745, Z    +0.000, E1   +58.469, E3 -255340.671}
SPL {X  -156.031, Y  +706.871, Z    +0.000, E1   +58.260, E3 -255349.816}
SPL {X  -154.558, Y  +712.835, Z    +0.000, E1   +58.028, E3 -255358.943}
SPL {X  -152.750, Y  +719.085, Z    +0.000, E1   +57.721, E3 -255368.790}
SPL {X  -150.741, Y  +725.111, Z    +0.000, E1   +57.387, E3 -255378.494}
SPL {X  -148.665, Y  +730.623, Z    +0.000, E1   +57.007, E3 -255387.642}
SPL {X  -146.664, Y  +735.425, Z    +0.000, E1   +56.657, E3 -255395.732}
SPL {X  -143.496, Y  +742.251, Z    +0.000, E1   +56.124, E3 -255407.426}
SPL {X  -140.752, Y  +747.564, Z    +0.000, E1   +55.554, E3 -255416.833}
SPL {X  -138.492, Y  +751.605, Z    +0.000, E1   +55.137, E3 -255424.024}
SPL {X  -124.324, Y  +772.199, Z    +0.000, E1   +48.708, E3 -255503.032}
ENDSPLINE

SPLINE
SPL {X  -129.118, Y  +765.975, Z    +0.000, E1   +43.713, E3 -255567.518}
SPL {X  -146.252, Y  +736.362, Z    +0.000, E1   +34.795, E3 -255616.695}
SPL {X  -155.916, Y  +707.374, Z    +0.000, E1   +22.878, E3 -255633.581}
SPL {X  -159.039, Y  +688.920, Z    +0.000, E1   +13.016, E3 -255638.815}
SPL {X  -159.777, Y  +679.762, Z    +0.000, E1    +7.372, E3 -255640.271}
SPL {X  -159.984, Y  +672.872, Z    +0.000, E1    +2.784, E3 -255640.867}
SPL {X  -159.990, Y  +668.898, Z    +0.000, E1    -0.346, E3 -255641.026}
SPL {X  -159.990, Y  +666.084, Z    +0.000, E1    -3.512, E3 -255641.148}
SPL {X  -159.990, Y  +662.904, Z    +0.000, E1    -7.618, E3 -255641.388}
SPL {X  -159.990, Y  +658.509, Z    +0.000, E1   -13.882, E3 -255641.923}
SPL {X  -159.990, Y  +652.317, Z    +0.000, E1   -22.778, E3 -255643.059}
SPL {X  -159.990, Y  +640.689, Z    +0.000, E1   -37.390, E3 -255644.601}
SPL {X  -159.990, Y  +585.634, Z    +0.000, E1   -68.681, E3 -255645.226}
SPL {X  -159.990, Y  +457.771, Z    +0.000, E1   -68.079, E3 -255735.787}
SPL {X  -159.990, Y  +453.218, Z    +0.000, E1   -67.322, E3 -255746.222}
SPL {X  -159.990, Y  +450.256, Z    +0.000, E1   -66.188, E3 -255758.155}
SPL {X  -159.990, Y  +445.667, Z    +0.000, E1   -65.356, E3 -255769.067}
SPL {X  -159.990, Y  +439.738, Z    +0.000, E1   -64.716, E3 -255779.879}
SPL {X  -159.990, Y  +433.217, Z    +0.000, E1   -63.756, E3 -255794.024}
SPL {X  -159.990, Y  +425.111, Z    +0.000, E1   -62.687, E3 -255810.564}
SPL {X  -159.990, Y  +418.218, Z    +0.000, E1   -61.769, E3 -255824.678}
SPL {X  -159.990, Y  +412.274, Z    +0.000, E1   -61.123, E3 -255836.082}
SPL {X  -159.990, Y  +408.631, Z    +0.000, E1   -60.233, E3 -255846.545}
SPL {X  -159.990, Y  +402.821, Z    +0.000, E1   -59.334, E3 -255860.072}
SPL {X  -159.990, Y  +395.849, Z    +0.000, E1   -58.799, E3 -255872.336}
SPL {X  -159.990, Y  +387.403, Z    +0.000, E1   -58.805, E3 -255883.182}
SPL {X  -159.948, Y  +378.844, Z    +0.000, E1   -58.798, E3 -255894.222}
SPL {X  -159.570, Y  +370.916, Z    +0.000, E1   -58.738, E3 -255904.818}
SPL {X  -158.865, Y  +363.563, Z    +0.000, E1   -58.615, E3 -255915.027}
SPL {X  -157.976, Y  +357.197, Z    +0.000, E1   -58.476, E3 -255924.128}
SPL {X  -156.730, Y  +350.368, Z    +0.000, E1   -58.276, E3 -255934.223}
SPL {X  -155.026, Y  +342.956, Z    +0.000, E1   -58.003, E3 -255945.495}
SPL {X  -152.946, Y  +335.551, Z    +0.000, E1   -57.653, E3 -255957.143}
SPL {X  -150.105, Y  +327.135, Z    +0.000, E1   -57.196, E3 -255970.763}
SPL {X  -146.578, Y  +318.377, Z    +0.000, E1   -56.572, E3 -255985.456}
SPL {X  -143.463, Y  +311.683, Z    +0.000, E1   -55.972, E3 -255997.070}
SPL {X  -140.858, Y  +306.633, Z    +0.000, E1   -55.477, E3 -256005.987}
SPL {X  -138.338, Y  +302.130, Z    +0.000, E1   -54.992, E3 -256014.037}
SPL {X  -124.427, Y  +281.929, Z    +0.000, E1   -46.852, E3 -256118.273}
ENDSPLINE

SPLINE
SPL {X  -148.251, Y  +322.346, Z    +0.000, E1   -33.039, E3 -256206.198}
SPL {X  -157.534, Y  +354.574, Z    +0.000, E1   -18.815, E3 -256223.027}
SPL {X  -159.548, Y  +370.614, Z    +0.000, E1    -9.656, E3 -256226.652}
SPL {X  -159.973, Y  +380.173, Z    +0.000, E1    -3.469, E3 -256227.719}
SPL {X  -159.990, Y  +384.078, Z    +0.000, E1    -0.490, E3 -256227.917}
SPL {X  -159.990, Y  +385.440, Z    +0.000, E1    +0.747, E3 -256227.958}
SPL {X  -159.990, Y  +388.179, Z    +0.000, E1    +3.660, E3 -256228.099}
SPL {X  -159.990, Y  +394.222, Z    +0.000, E1   +11.674, E3 -256228.692}
SPL {X  -159.990, Y  +403.976, Z    +0.000, E1   +25.456, E3 -256230.571}
SPL {X  -159.990, Y  +417.120, Z    +0.000, E1   +39.678, E3 -256234.603}
SPL {X  -159.990, Y  +456.927, Z    +0.000, E1   +55.382, E3 -256256.463}
SPL {X  -159.990, Y  +530.047, Z    +0.000, E1   +58.901, E3 -256326.297}
SPL {X  -159.990, Y  +538.035, Z    +0.000, E1   +58.900, E3 -256336.522}
SPL {X  -159.990, Y  +546.883, Z    +0.000, E1   +58.912, E3 -256347.826}
SPL {X  -159.990, Y  +555.949, Z    +0.000, E1   +58.900, E3 -256359.445}
SPL {X  -159.990, Y  +563.718, Z    +0.000, E1   +58.903, E3 -256369.366}
SPL {X  -159.990, Y  +571.529, Z    +0.000, E1   +58.906, E3 -256379.350}
SPL {X  -159.990, Y  +579.859, Z    +0.000, E1   +58.907, E3 -256390.009}
SPL {X  -159.990, Y  +588.526, Z    +0.000, E1   +58.910, E3 -256401.083}
SPL {X  -159.990, Y  +596.521, Z    +0.000, E1   +58.902, E3 -256411.342}
SPL {X  -159.990, Y  +605.444, Z    +0.000, E1   +58.918, E3 -256422.731}
SPL {X  -159.990, Y  +618.101, Z    +0.000, E1   +58.946, E3 -256438.878}
SPL {X  -159.990, Y  +629.920, Z    +0.000, E1   +58.912, E3 -256454.071}
SPL {X  -159.990, Y  +638.424, Z    +0.000, E1   +58.901, E3 -256464.971}
SPL {X  -159.990, Y  +645.995, Z    +0.000, E1   +58.900, E3 -256474.659}
SPL {X  -159.990, Y  +654.206, Z    +0.000, E1   +58.908, E3 -256485.150}
SPL {X  -159.990, Y  +661.562, Z    +0.000, E1   +58.900, E3 -256494.578}
SPL {X  -159.990, Y  +670.328, Z    +0.000, E1   +58.911, E3 -256505.777}
SPL {X  -159.795, Y  +679.404, Z    +0.000, E1   +58.876, E3 -256517.602}
SPL {X  -159.282, Y  +686.534, Z    +0.000, E1   +58.787, E3 -256527.276}
SPL {X  -158.463, Y  +693.553, Z    +0.000, E1   +58.665, E3 -256537.117}
SPL {X  -157.294, Y  +700.745, Z    +0.000, E1   +58.469, E3 -256547.567}
SPL {X  -156.031, Y  +706.871, Z    +0.000, E1   +58.260, E3 -256556.713}
SPL {X  -154.558, Y  +712.835, Z    +0.000, E1   +58.028, E3 -256565.840}
SPL {X  -152.750, Y  +719.085, Z    +0.000, E1   +57.721, E3 -256575.686}
SPL {X  -150.741, Y  +725.111, Z    +0.000, E1   +57.387, E3 -256585.390}
SPL {X  -148.665, Y  +730.623, Z    +0.000, E1   +57.007, E3 -256594.539}
SPL {X  -146.664, Y  +735.425, Z    +0.000, E1   +56.657, E3 -256602.629}
SPL {X  -143.496, Y  +742.251, Z    +0.000, E1   +56.124, E3 -256614.322}
SPL {X  -140.752, Y  +747.564, Z    +0.000, E1   +55.554, E3 -256623.730}
SPL {X  -138.492, Y  +751.605, Z    +0.000, E1   +55.137, E3 -256630.921}
SPL {X  -124.324, Y  +772.199, Z    +0.000, E1   +48.708, E3 -256709.929}
ENDSPLINE

SPLINE
SPL {X  -129.118, Y  +765.975, Z    +0.000, E1   +43.713, E3 -256774.414}
SPL {X  -146.252, Y  +736.362, Z    +0.000, E1   +34.795, E3 -256823.592}
SPL {X  -155.916, Y  +707.374, Z    +0.000, E1   +22.878, E3 -256840.477}
SPL {X  -159.039, Y  +688.920, Z    +0.000, E1   +13.016, E3 -256845.712}
SPL {X  -159.888, Y  +677.224, Z    +0.000, E1    +5.773, E3 -256847.425}
SPL {X  -159.990, Y  +671.755, Z    +0.000, E1    +1.905, E3 -256847.828}
SPL {X  -159.990, Y  +669.598, Z    +0.000, E1    +0.205, E3 -256847.901}
SPL {X  -159.990, Y  +667.097, Z    +0.000, E1    -2.190, E3 -256847.996}
SPL {X  -159.990, Y  +662.904, Z    +0.000, E1    -7.618, E3 -256848.284}
SPL {X  -159.990, Y  +658.509, Z    +0.000, E1   -13.882, E3 -256848.820}
SPL {X  -159.990, Y  +652.317, Z    +0.000, E1   -22.778, E3 -256849.955}
SPL {X  -159.990, Y  +640.689, Z    +0.000, E1   -37.390, E3 -256851.498}
SPL {X  -159.990, Y  +585.634, Z    +0.000, E1   -68.681, E3 -256852.122}
SPL {X  -159.990, Y  +457.771, Z    +0.000, E1   -68.079, E3 -256942.683}
SPL {X  -159.990, Y  +453.218, Z    +0.000, E1   -67.322, E3 -256953.119}
SPL {X  -159.990, Y  +450.256, Z    +0.000, E1   -66.188, E3 -256965.051}
SPL {X  -159.990, Y  +445.667, Z    +0.000, E1   -65.356, E3 -256975.963}
SPL {X  -159.990, Y  +439.738, Z    +0.000, E1   -64.716, E3 -256986.776}
SPL {X  -159.990, Y  +435.528, Z    +0.000, E1   -63.972, E3 -256996.652}
SPL {X  -159.990, Y  +429.021, Z    +0.000, E1   -63.228, E3 -257009.264}
SPL {X  -159.990, Y  +423.267, Z    +0.000, E1   -62.365, E3 -257021.562}
SPL {X  -159.990, Y  +418.218, Z    +0.000, E1   -61.769, E3 -257031.575}
SPL {X  -159.990, Y  +412.274, Z    +0.000, E1   -61.123, E3 -257042.979}
SPL {X  -159.990, Y  +408.631, Z    +0.000, E1   -60.233, E3 -257053.441}
SPL {X  -159.990, Y  +404.834, Z    +0.000, E1   -59.529, E3 -257062.896}
SPL {X  -159.990, Y  +397.866, Z    +0.000, E1   -58.924, E3 -257075.984}
SPL {X  -159.990, Y  +387.403, Z    +0.000, E1   -58.805, E3 -257090.079}
SPL {X  -159.948, Y  +378.844, Z    +0.000, E1   -58.798, E3 -257101.119}
SPL {X  -159.570, Y  +370.916, Z    +0.000, E1   -58.738, E3 -257111.714}
SPL {X  -158.865, Y  +363.563, Z    +0.000, E1   -58.615, E3 -257121.923}
SPL {X  -157.976, Y  +357.197, Z    +0.000, E1   -58.476, E3 -257131.024}
SPL {X  -156.730, Y  +350.368, Z    +0.000, E1   -58.276, E3 -257141.120}
SPL {X  -155.026, Y  +342.956, Z    +0.000, E1   -58.003, E3 -257152.392}
SPL {X  -152.946, Y  +335.551, Z    +0.000, E1   -57.653, E3 -257164.040}
SPL {X  -150.105, Y  +327.135, Z    +0.000, E1   -57.196, E3 -257177.660}
SPL {X  -146.578, Y  +318.377, Z    +0.000, E1   -56.572, E3 -257192.353}
SPL {X  -143.463, Y  +311.683, Z    +0.000, E1   -55.972, E3 -257203.966}
SPL {X  -140.858, Y  +306.633, Z    +0.000, E1   -55.477, E3 -257212.884}
SPL {X  -138.338, Y  +302.130, Z    +0.000, E1   -54.992, E3 -257220.933}
SPL {X  -124.427, Y  +281.929, Z    +0.000, E1   -46.852, E3 -257325.169}
ENDSPLINE

SPLINE
SPL {X  -148.251, Y  +322.346, Z    +0.000, E1   -33.039, E3 -257413.095}
SPL {X  -157.534, Y  +354.574, Z    +0.000, E1   -18.815, E3 -257429.924}
SPL {X  -159.548, Y  +370.614, Z    +0.000, E1    -9.656, E3 -257433.549}
SPL {X  -159.928, Y  +378.035, Z    +0.000, E1    -4.866, E3 -257434.465}
SPL {X  -159.990, Y  +383.381, Z    +0.000, E1    -1.123, E3 -257434.785}
SPL {X  -159.990, Y  +386.348, Z    +0.000, E1    +1.571, E3 -257434.894}
SPL {X  -159.990, Y  +391.422, Z    +0.000, E1    +7.757, E3 -257435.268}
SPL {X  -159.990, Y  +399.099, Z    +0.000, E1   +18.787, E3 -257436.375}
SPL {X  -159.990, Y  +406.316, Z    +0.000, E1   +28.569, E3 -257438.052}
SPL {X  -159.990, Y  +417.120, Z    +0.000, E1   +39.678, E3 -257441.499}
SPL {X  -159.990, Y  +456.927, Z    +0.000, E1   +55.382, E3 -257463.360}
SPL {X  -159.990, Y  +530.047, Z    +0.000, E1   +58.901, E3 -257533.194}
SPL {X  -159.990, Y  +538.035, Z    +0.000, E1   +58.900, E3 -257543.419}
SPL {X  -159.990, Y  +546.883, Z    +0.000, E1   +58.912, E3 -257554.723}
SPL {X  -159.990, Y  +555.949, Z    +0.000, E1   +58.900, E3 -257566.342}
SPL {X  -159.990, Y  +563.718, Z    +0.000, E1   +58.903, E3 -257576.262}
SPL {X  -159.990, Y  +571.529, Z    +0.000, E1   +58.906, E3 -257586.246}
SPL {X  -159.990, Y  +579.859, Z    +0.000, E1   +58.907, E3 -257596.906}
SPL {X  -159.990, Y  +588.526, Z    +0.000, E1   +58.910, E3 -257607.979}
SPL {X  -159.990, Y  +596.521, Z    +0.000, E1   +58.902, E3 -257618.238}
SPL {X  -159.990, Y  +605.444, Z    +0.000, E1   +58.918, E3 -257629.628}
SPL {X  -159.990, Y  +618.101, Z    +0.000, E1   +58.946, E3 -257645.775}
SPL {X  -159.990, Y  +629.920, Z    +0.000, E1   +58.912, E3 -257660.968}
SPL {X  -159.990, Y  +638.424, Z    +0.000, E1   +58.901, E3 -257671.868}
SPL {X  -159.990, Y  +645.995, Z    +0.000, E1   +58.900, E3 -257681.555}
SPL {X  -159.990, Y  +654.206, Z    +0.000, E1   +58.908, E3 -257692.046}
SPL {X  -159.990, Y  +661.562, Z    +0.000, E1   +58.900, E3 -257701.474}
SPL {X  -159.990, Y  +670.328, Z    +0.000, E1   +58.911, E3 -257712.673}
SPL {X  -159.795, Y  +679.404, Z    +0.000, E1   +58.876, E3 -257724.499}
SPL {X  -159.282, Y  +686.534, Z    +0.000, E1   +58.787, E3 -257734.173}
SPL {X  -158.463, Y  +693.553, Z    +0.000, E1   +58.665, E3 -257744.014}
SPL {X  -157.294, Y  +700.745, Z    +0.000, E1   +58.469, E3 -257754.464}
SPL {X  -156.031, Y  +706.871, Z    +0.000, E1   +58.260, E3 -257763.609}
SPL {X  -154.558, Y  +712.835, Z    +0.000, E1   +58.028, E3 -257772.737}
SPL {X  -152.750, Y  +719.085, Z    +0.000, E1   +57.721, E3 -257782.583}
SPL {X  -150.741, Y  +725.111, Z    +0.000, E1   +57.387, E3 -257792.287}
SPL {X  -148.665, Y  +730.623, Z    +0.000, E1   +57.007, E3 -257801.435}
SPL {X  -146.664, Y  +735.425, Z    +0.000, E1   +56.657, E3 -257809.525}
SPL {X  -143.496, Y  +742.251, Z    +0.000, E1   +56.124, E3 -257821.219}
SPL {X  -140.752, Y  +747.564, Z    +0.000, E1   +55.554, E3 -257830.626}
SPL {X  -138.492, Y  +751.605, Z    +0.000, E1   +55.137, E3 -257837.817}
SPL {X  -124.324, Y  +772.199, Z    +0.000, E1   +48.708, E3 -257916.825}
ENDSPLINE

SPLINE
SPL {X  -129.118, Y  +765.975, Z    +0.000, E1   +43.713, E3 -257981.311}
SPL {X  -146.252, Y  +736.362, Z    +0.000, E1   +34.795, E3 -258030.488}
SPL {X  -154.088, Y  +714.555, Z    +0.000, E1   +26.177, E3 -258044.505}
SPL {X  -156.688, Y  +703.837, Z    +0.000, E1   +21.096, E3 -258048.676}
SPL {X  -159.039, Y  +688.920, Z    +0.000, E1   +13.016, E3 -258052.608}
SPL {X  -159.888, Y  +677.224, Z    +0.000, E1    +5.773, E3 -258054.321}
SPL {X  -159.990, Y  +670.275, Z    +0.000, E1    +0.854, E3 -258054.775}
SPL {X  -159.990, Y  +667.097, Z    +0.000, E1    -2.190, E3 -258054.893}
SPL {X  -159.990, Y  +662.904, Z    +0.000, E1    -7.618, E3 -258055.181}
SPL {X  -159.990, Y  +658.509, Z    +0.000, E1   -13.882, E3 -258055.716}
SPL {X  -159.990, Y  +652.317, Z    +0.000, E1   -22.778, E3 -258056.852}
SPL {X  -159.990, Y  +640.689, Z    +0.000, E1   -37.390, E3 -258058.394}
SPL {X  -159.990, Y  +585.634, Z    +0.000, E1   -68.681, E3 -258059.019}
SPL {X  -159.990, Y  +457.771, Z    +0.000, E1   -68.079, E3 -258149.580}
SPL {X  -159.990, Y  +453.218, Z    +0.000, E1   -67.322, E3 -258160.015}
SPL {X  -159.990, Y  +450.256, Z    +0.000, E1   -66.188, E3 -258171.948}
SPL {X  -159.990, Y  +445.667, Z    +0.000, E1   -65.356, E3 -258182.860}
SPL {X  -159.990, Y  +439.738, Z    +0.000, E1   -64.716, E3 -258193.672}
SPL {X  -159.990, Y  +435.528, Z    +0.000, E1   -63.972, E3 -258203.548}
SPL {X  -159.990, Y  +429.021, Z    +0.000, E1   -63.228, E3 -258216.161}
SPL {X  -159.990, Y  +423.267, Z    +0.000, E1   -62.365, E3 -258228.459}
SPL {X  -159.990, Y  +418.218, Z    +0.000, E1   -61.769, E3 -258238.471}
SPL {X  -159.990, Y  +412.274, Z    +0.000, E1   -61.123, E3 -258249.875}
SPL {X  -159.990, Y  +408.631, Z    +0.000, E1   -60.233, E3 -258260.338}
SPL {X  -159.990, Y  +404.834, Z    +0.000, E1   -59.529, E3 -258269.793}
SPL {X  -159.990, Y  +397.866, Z    +0.000, E1   -58.924, E3 -258282.880}
SPL {X  -159.990, Y  +387.403, Z    +0.000, E1   -58.805, E3 -258296.975}
SPL {X  -159.948, Y  +378.844, Z    +0.000, E1   -58.798, E3 -258308.015}
SPL {X  -159.570, Y  +370.916, Z    +0.000, E1   -58.738, E3 -258318.611}
SPL {X  -158.865, Y  +363.563, Z    +0.000, E1   -58.615, E3 -258328.820}
SPL {X  -157.976, Y  +357.197, Z    +0.000, E1   -58.476, E3 -258337.921}
SPL {X  -156.730, Y  +350.368, Z    +0.000, E1   -58.276, E3 -258348.016}
SPL {X  -155.026, Y  +342.956, Z    +0.000, E1   -58.003, E3 -258359.288}
SPL {X  -152.946, Y  +335.551, Z    +0.000, E1   -57.653, E3 -258370.936}
SPL {X  -150.899, Y  +329.336, Z    +0.000, E1   -57.290, E3 -258381.002}
SPL {X  -149.179, Y  +324.687, Z    +0.000, E1   -56.983, E3 -258388.691}
SPL {X  -146.578, Y  +318.377, Z    +0.000, E1   -56.572, E3 -258399.249}
SPL {X  -143.463, Y  +311.683, Z    +0.000, E1   -55.972, E3 -258410.863}
SPL {X  -140.858, Y  +306.633, Z    +0.000, E1   -55.477, E3 -258419.780}
SPL {X  -138.338, Y  +302.130, Z    +0.000, E1   -54.992, E3 -258427.830}
SPL {X  -124.427, Y  +281.929, Z    +0.000, E1   -46.852, E3 -258532.066}
ENDSPLINE

SPLINE
SPL {X  -138.506, Y  +302.419, Z    +0.000, E1   -39.451, E3 -258598.040}
SPL {X  -149.686, Y  +326.013, Z    +0.000, E1   -31.658, E3 -258623.177}
SPL {X  -156.481, Y  +349.177, Z    +0.000, E1   -21.514, E3 -258635.174}
SPL {X  -159.327, Y  +367.953, Z    +0.000, E1   -11.342, E3 -258639.965}
SPL {X  -159.973, Y  +380.173, Z    +0.000, E1    -3.469, E3 -258641.513}
SPL {X  -159.990, Y  +384.078, Z    +0.000, E1    -0.490, E3 -258641.710}
SPL {X  -159.990, Y  +385.440, Z    +0.000, E1    +0.747, E3 -258641.751}
SPL {X  -159.990, Y  +388.179, Z    +0.000, E1    +3.660, E3 -258641.892}
SPL {X  -159.990, Y  +394.222, Z    +0.000, E1   +11.674, E3 -258642.485}
SPL {X  -159.990, Y  +403.976, Z    +0.000, E1   +25.456, E3 -258644.364}
SPL {X  -159.990, Y  +417.120, Z    +0.000, E1   +39.678, E3 -258648.396}
SPL {X  -159.990, Y  +456.927, Z    +0.000, E1   +55.382, E3 -258670.256}
SPL {X  -159.990, Y  +530.047, Z    +0.000, E1   +58.901, E3 -258740.090}
SPL {X  -159.990, Y  +538.035, Z    +0.000, E1   +58.900, E3 -258750.316}
SPL {X  -159.990, Y  +546.883, Z    +0.000, E1   +58.912, E3 -258761.619}
SPL {X  -159.990, Y  +555.949, Z    +0.000, E1   +58.900, E3 -258773.239}
SPL {X  -159.990, Y  +563.718, Z    +0.000, E1   +58.903, E3 -258783.159}
SPL {X  -159.990, Y  +571.529, Z    +0.000, E1   +58.906, E3 -258793.143}
SPL {X  -159.990, Y  +579.859, Z    +0.000, E1   +58.907, E3 -258803.802}
SPL {X  -159.990, Y  +588.526, Z    +0.000, E1   +58.910, E3 -258814.876}
SPL {X  -159.990, Y  +596.521, Z    +0.000, E1   +58.902, E3 -258825.135}
SPL {X  -159.990, Y  +605.444, Z    +0.000, E1   +58.918, E3 -258836.524}
SPL {X  -159.990, Y  +613.908, Z    +0.000, E1   +58.900, E3 -258847.383}
SPL {X  -159.990, Y  +621.342, Z    +0.000, E1   +58.904, E3 -258856.892}
SPL {X  -159.990, Y  +629.920, Z    +0.000, E1   +58.912, E3 -258867.864}
SPL {X  -159.990, Y  +642.398, Z    +0.000, E1   +58.947, E3 -258883.772}
SPL {X  -159.990, Y  +654.206, Z    +0.000, E1   +58.908, E3 -258898.943}
SPL {X  -159.990, Y  +661.562, Z    +0.000, E1   +58.900, E3 -258908.371}
SPL {X  -159.990, Y  +670.328, Z    +0.000, E1   +58.911, E3 -258919.570}
SPL {X  -159.795, Y  +679.404, Z    +0.000, E1   +58.876, E3 -258931.395}
SPL {X  -159.282, Y  +686.534, Z    +0.000, E1   +58.787, E3 -258941.069}
SPL {X  -158.463, Y  +693.553, Z    +0.000, E1   +58.665, E3 -258950.910}
SPL {X  -157.294, Y  +700.745, Z    +0.000, E1   +58.469, E3 -258961.360}
SPL {X  -156.031, Y  +706.871, Z    +0.000, E1   +58.260, E3 -258970.506}
SPL {X  -154.558, Y  +712.835, Z    +0.000, E1   +58.028, E3 -258979.633}
SPL {X  -152.750, Y  +719.085, Z    +0.000, E1   +57.721, E3 -258989.479}
SPL {X  -150.741, Y  +725.111, Z    +0.000, E1   +57.387, E3 -258999.183}
SPL {X  -148.665, Y  +730.623, Z    +0.000, E1   +57.007, E3 -259008.332}
SPL {X  -146.664, Y  +735.425, Z    +0.000, E1   +56.657, E3 -259016.422}
SPL {X  -143.496, Y  +742.251, Z    +0.000, E1   +56.124, E3 -259028.115}
SPL {X  -140.752, Y  +747.564, Z    +0.000, E1   +55.554, E3 -259037.523}
SPL {X  -138.492, Y  +751.605, Z    +0.000, E1   +55.137, E3 -259044.714}
SPL {X  -124.324, Y  +772.199, Z    +0.000, E1   +48.708, E3 -259123.722}
ENDSPLINE

SPLINE
SPL {X  -129.118, Y  +765.975, Z    +0.000, E1   +43.713, E3 -259188.207}
SPL {X  -146.252, Y  +736.362, Z    +0.000, E1   +34.795, E3 -259237.385}
SPL {X  -154.088, Y  +714.555, Z    +0.000, E1   +26.177, E3 -259251.401}
SPL {X  -156.688, Y  +703.837, Z    +0.000, E1   +21.096, E3 -259255.573}
SPL {X  -159.039, Y  +688.920, Z    +0.000, E1   +13.016, E3 -259259.505}
SPL {X  -159.888, Y  +677.224, Z    +0.000, E1    +5.773, E3 -259261.218}
SPL {X  -159.990, Y  +671.755, Z    +0.000, E1    +1.905, E3 -259261.621}
SPL {X  -159.990, Y  +669.598, Z    +0.000, E1    +0.205, E3 -259261.694}
SPL {X  -159.990, Y  +667.097, Z    +0.000, E1    -2.190, E3 -259261.789}
SPL {X  -159.990, Y  +662.904, Z    +0.000, E1    -7.618, E3 -259262.077}
SPL {X  -159.990, Y  +658.509, Z    +0.000, E1   -13.882, E3 -259262.613}
SPL {X  -159.990, Y  +652.317, Z    +0.000, E1   -22.778, E3 -259263.748}
SPL {X  -159.990, Y  +641.893, Z    +0.000, E1   -35.310, E3 -259266.713}
SPL {X  -159.990, Y  +636.123, Z    +0.000, E1   -46.139, E3 -259259.778}
SPL {X  -159.990, Y  +585.634, Z    +0.000, E1   -68.681, E3 -259265.915}
SPL {X  -159.990, Y  +457.771, Z    +0.000, E1   -68.079, E3 -259356.476}
SPL {X  -159.990, Y  +453.218, Z    +0.000, E1   -67.322, E3 -259366.912}
SPL {X  -159.990, Y  +450.256, Z    +0.000, E1   -66.188, E3 -259378.844}
SPL {X  -159.990, Y  +445.667, Z    +0.000, E1   -65.356, E3 -259389.756}
SPL {X  -159.990, Y  +439.738, Z    +0.000, E1   -64.716, E3 -259400.569}
SPL {X  -159.990, Y  +435.528, Z    +0.000, E1   -63.972, E3 -259410.445}
SPL {X  -159.990, Y  +429.021, Z    +0.000, E1   -63.228, E3 -259423.058}
SPL {X  -159.990, Y  +423.267, Z    +0.000, E1   -62.365, E3 -259435.356}
SPL {X  -159.990, Y  +418.218, Z    +0.000, E1   -61.769, E3 -259445.368}
SPL {X  -159.990, Y  +412.274, Z    +0.000, E1   -61.123, E3 -259456.772}
SPL {X  -159.990, Y  +408.631, Z    +0.000, E1   -60.233, E3 -259467.234}
SPL {X  -159.990, Y  +404.834, Z    +0.000, E1   -59.529, E3 -259476.689}
SPL {X  -159.990, Y  +397.866, Z    +0.000, E1   -58.924, E3 -259489.777}
SPL {X  -159.990, Y  +387.403, Z    +0.000, E1   -58.805, E3 -259503.872}
SPL {X  -159.948, Y  +378.844, Z    +0.000, E1   -58.798, E3 -259514.912}
SPL {X  -159.570, Y  +370.916, Z    +0.000, E1   -58.738, E3 -259525.507}
SPL {X  -158.865, Y  +363.563, Z    +0.000, E1   -58.615, E3 -259535.717}
SPL {X  -157.976, Y  +357.197, Z    +0.000, E1   -58.476, E3 -259544.817}
SPL {X  -156.730, Y  +350.368, Z    +0.000, E1   -58.276, E3 -259554.913}
SPL {X  -155.026, Y  +342.956, Z    +0.000, E1   -58.003, E3 -259566.185}
SPL {X  -152.946, Y  +335.551, Z    +0.000, E1   -57.653, E3 -259577.833}
SPL {X  -150.899, Y  +329.336, Z    +0.000, E1   -57.290, E3 -259587.898}
SPL {X  -149.179, Y  +324.687, Z    +0.000, E1   -56.983, E3 -259595.588}
SPL {X  -147.281, Y  +320.009, Z    +0.000, E1   -56.662, E3 -259603.414}
SPL {X  -144.114, Y  +313.017, Z    +0.000, E1   -56.131, E3 -259615.381}
SPL {X  -140.858, Y  +306.633, Z    +0.000, E1   -55.477, E3 -259626.677}
SPL {X  -138.338, Y  +302.130, Z    +0.000, E1   -54.992, E3 -259634.726}
SPL {X  -124.427, Y  +281.929, Z    +0.000, E1   -46.852, E3 -259738.963}
ENDSPLINE

SPLINE
SPL {X  -148.251, Y  +322.346, Z    +0.000, E1   -33.039, E3 -259826.888}
SPL {X  -157.534, Y  +354.574, Z    +0.000, E1   -18.815, E3 -259843.717}
SPL {X  -159.548, Y  +370.614, Z    +0.000, E1    -9.656, E3 -259847.342}
SPL {X  -159.928, Y  +378.035, Z    +0.000, E1    -4.866, E3 -259848.258}
SPL {X  -159.990, Y  +383.381, Z    +0.000, E1    -1.123, E3 -259848.578}
SPL {X  -159.990, Y  +386.348, Z    +0.000, E1    +1.571, E3 -259848.687}
SPL {X  -159.990, Y  +391.422, Z    +0.000, E1    +7.757, E3 -259849.062}
SPL {X  -159.990, Y  +396.843, Z    +0.000, E1   +15.720, E3 -259849.723}
SPL {X  -159.990, Y  +403.976, Z    +0.000, E1   +25.456, E3 -259851.261}
SPL {X  -159.990, Y  +417.120, Z    +0.000, E1   +39.678, E3 -259855.292}
SPL {X  -159.990, Y  +456.927, Z    +0.000, E1   +55.382, E3 -259877.153}
SPL {X  -159.990, Y  +530.047, Z    +0.000, E1   +58.901, E3 -259946.987}
SPL {X  -159.990, Y  +538.035, Z    +0.000, E1   +58.900, E3 -259957.212}
SPL {X  -159.990, Y  +546.883, Z    +0.000, E1   +58.912, E3 -259968.516}
SPL {X  -159.990, Y  +555.949, Z    +0.000, E1   +58.900, E3 -259980.135}
SPL {X  -159.990, Y  +563.718, Z    +0.000, E1   +58.903, E3 -259990.055}
SPL {X  -159.990, Y  +571.529, Z    +0.000, E1   +58.906, E3 -260000.039}
SPL {X  -159.990, Y  +579.859, Z    +0.000, E1   +58.907, E3 -260010.699}
SPL {X  -159.990, Y  +588.526, Z    +0.000, E1   +58.910, E3 -260021.772}
SPL {X  -159.990, Y  +596.521, Z    +0.000, E1   +58.902, E3 -260032.031}
SPL {X  -159.990, Y  +605.444, Z    +0.000, E1   +58.918, E3 -260043.421}
SPL {X  -159.990, Y  +618.101, Z    +0.000, E1   +58.946, E3 -260059.568}
SPL {X  -159.990, Y  +629.920, Z    +0.000, E1   +58.912, E3 -260074.761}
SPL {X  -159.990, Y  +638.424, Z    +0.000, E1   +58.901, E3 -260085.661}
SPL {X  -159.990, Y  +645.995, Z    +0.000, E1   +58.900, E3 -260095.349}
SPL {X  -159.990, Y  +654.206, Z    +0.000, E1   +58.908, E3 -260105.839}
SPL {X  -159.990, Y  +661.562, Z    +0.000, E1   +58.900, E3 -260115.267}
SPL {X  -159.990, Y  +670.328, Z    +0.000, E1   +58.911, E3 -260126.467}
SPL {X  -159.795, Y  +679.404, Z    +0.000, E1   +58.876, E3 -260138.292}
SPL {X  -159.282, Y  +686.534, Z    +0.000, E1   +58.787, E3 -260147.966}
SPL {X  -158.463, Y  +693.553, Z    +0.000, E1   +58.665, E3 -260157.807}
SPL {X  -157.294, Y  +700.745, Z    +0.000, E1   +58.469, E3 -260168.257}
SPL {X  -156.031, Y  +706.871, Z    +0.000, E1   +58.260, E3 -260177.402}
SPL {X  -154.558, Y  +712.835, Z    +0.000, E1   +58.028, E3 -260186.530}
SPL {X  -152.750, Y  +719.085, Z    +0.000, E1   +57.721, E3 -260196.376}
SPL {X  -150.741, Y  +725.111, Z    +0.000, E1   +57.387, E3 -260206.080}
SPL {X  -148.665, Y  +730.623, Z    +0.000, E1   +57.007, E3 -260215.229}
SPL {X  -146.664, Y  +735.425, Z    +0.000, E1   +56.657, E3 -260223.319}
SPL {X  -143.496, Y  +742.251, Z    +0.000, E1   +56.124, E3 -260235.012}
SPL {X  -140.752, Y  +747.564, Z    +0.000, E1   +55.554, E3 -260244.419}
SPL {X  -138.492, Y  +751.605, Z    +0.000, E1   +55.137, E3 -260251.610}
SPL {X  -124.324, Y  +772.199, Z    +0.000, E1   +48.708, E3 -260330.618}
ENDSPLINE

SPLINE
SPL {X  -129.118, Y  +765.975, Z    +0.000, E1   +43.713, E3 -260395.104}
SPL {X  -146.252, Y  +736.362, Z    +0.000, E1   +34.795, E3 -260444.282}
SPL {X  -155.916, Y  +707.374, Z    +0.000, E1   +22.878, E3 -260461.167}
SPL {X  -159.039, Y  +688.920, Z    +0.000, E1   +13.016, E3 -260466.402}
SPL {X  -159.777, Y  +679.762, Z    +0.000, E1    +7.372, E3 -260467.857}
SPL {X  -159.984, Y  +672.872, Z    +0.000, E1    +2.784, E3 -260468.454}
SPL {X  -159.990, Y  +669.598, Z    +0.000, E1    +0.205, E3 -260468.591}
SPL {X  -159.990, Y  +667.097, Z    +0.000, E1    -2.190, E3 -260468.686}
SPL {X  -159.990, Y  +662.904, Z    +0.000, E1    -7.618, E3 -260468.974}
SPL {X  -159.990, Y  +658.509, Z    +0.000, E1   -13.882, E3 -260469.510}
SPL {X  -159.990, Y  +652.317, Z    +0.000, E1   -22.778, E3 -260470.645}
SPL {X  -159.990, Y  +640.689, Z    +0.000, E1   -37.390, E3 -260472.188}
SPL {X  -159.990, Y  +585.634, Z    +0.000, E1   -68.681, E3 -260472.812}
SPL {X  -159.990, Y  +457.771, Z    +0.000, E1   -68.079, E3 -260563.373}
SPL {X  -159.990, Y  +453.218, Z    +0.000, E1   -67.322, E3 -260573.808}
SPL {X  -159.990, Y  +450.256, Z    +0.000, E1   -66.188, E3 -260585.741}
SPL {X  -159.990, Y  +445.667, Z    +0.000, E1   -65.356, E3 -260596.653}
SPL {X  -159.990, Y  +439.738, Z    +0.000, E1   -64.716, E3 -260607.466}
SPL {X  -159.990, Y  +435.528, Z    +0.000, E1   -63.972, E3 -260617.341}
SPL {X  -159.990, Y  +429.021, Z    +0.000, E1   -63.228, E3 -260629.954}
SPL {X  -159.990, Y  +423.267, Z    +0.000, E1   -62.365, E3 -260642.252}
SPL {X  -159.990, Y  +418.218, Z    +0.000, E1   -61.769, E3 -260652.265}
SPL {X  -159.990, Y  +412.274, Z    +0.000, E1   -61.123, E3 -260663.669}
SPL {X  -159.990, Y  +408.631, Z    +0.000, E1   -60.233, E3 -260674.131}
SPL {X  -159.990, Y  +402.821, Z    +0.000, E1   -59.334, E3 -260687.658}
SPL {X  -159.990, Y  +395.849, Z    +0.000, E1   -58.799, E3 -260699.922}
SPL {X  -159.990, Y  +387.403, Z    +0.000, E1   -58.805, E3 -260710.769}
SPL {X  -159.948, Y  +378.844, Z    +0.000, E1   -58.798, E3 -260721.808}
SPL {X  -159.570, Y  +370.916, Z    +0.000, E1   -58.738, E3 -260732.404}
SPL {X  -158.865, Y  +363.563, Z    +0.000, E1   -58.615, E3 -260742.613}
SPL {X  -157.976, Y  +357.197, Z    +0.000, E1   -58.476, E3 -260751.714}
SPL {X  -156.730, Y  +350.368, Z    +0.000, E1   -58.276, E3 -260761.809}
SPL {X  -155.026, Y  +342.956, Z    +0.000, E1   -58.003, E3 -260773.081}
SPL {X  -152.946, Y  +335.551, Z    +0.000, E1   -57.653, E3 -260784.729}
SPL {X  -150.105, Y  +327.135, Z    +0.000, E1   -57.196, E3 -260798.349}
SPL {X  -146.578, Y  +318.377, Z    +0.000, E1   -56.572, E3 -260813.042}
SPL {X  -143.463, Y  +311.683, Z    +0.000, E1   -55.972, E3 -260824.656}
SPL {X  -140.858, Y  +306.633, Z    +0.000, E1   -55.477, E3 -260833.573}
SPL {X  -138.338, Y  +302.130, Z    +0.000, E1   -54.992, E3 -260841.623}
SPL {X  -124.427, Y  +281.929, Z    +0.000, E1   -46.852, E3 -260945.859}
ENDSPLINE

SPLINE
SPL {X  -148.251, Y  +322.346, Z    +0.000, E1   -33.039, E3 -261033.784}
SPL {X  -156.481, Y  +349.177, Z    +0.000, E1   -21.514, E3 -261048.967}
SPL {X  -159.327, Y  +367.953, Z    +0.000, E1   -11.342, E3 -261053.759}
SPL {X  -159.973, Y  +380.173, Z    +0.000, E1    -3.469, E3 -261055.306}
SPL {X  -159.990, Y  +384.078, Z    +0.000, E1    -0.490, E3 -261055.503}
SPL {X  -159.990, Y  +385.440, Z    +0.000, E1    +0.747, E3 -261055.544}
SPL {X  -159.990, Y  +388.179, Z    +0.000, E1    +3.660, E3 -261055.685}
SPL {X  -159.990, Y  +394.222, Z    +0.000, E1   +11.674, E3 -261056.278}
SPL {X  -159.990, Y  +403.976, Z    +0.000, E1   +25.456, E3 -261058.158}
SPL {X  -159.990, Y  +417.120, Z    +0.000, E1   +39.678, E3 -261062.189}
SPL {X  -159.990, Y  +456.927, Z    +0.000, E1   +55.382, E3 -261084.049}
SPL {X  -159.990, Y  +530.047, Z    +0.000, E1   +58.901, E3 -261153.883}
SPL {X  -159.990, Y  +538.035, Z    +0.000, E1   +58.900, E3 -261164.109}
SPL {X  -159.990, Y  +546.883, Z    +0.000, E1   +58.912, E3 -261175.412}
SPL {X  -159.990, Y  +555.949, Z    +0.000, E1   +58.900, E3 -261187.032}
SPL {X  -159.990, Y  +563.718, Z    +0.000, E1   +58.903, E3 -261196.952}
SPL {X  -159.990, Y  +571.529, Z    +0.000, E1   +58.906, E3 -261206.936}
SPL {X  -159.990, Y  +579.859, Z    +0.000, E1   +58.907, E3 -261217.595}
SPL {X  -159.990, Y  +588.526, Z    +0.000, E1   +58.910, E3 -261228.669}
SPL {X  -159.990, Y  +596.521, Z    +0.000, E1   +58.902, E3 -261238.928}
SPL {X  -159.990, Y  +605.444, Z    +0.000, E1   +58.918, E3 -261250.317}
SPL {X  -159.990, Y  +613.908, Z    +0.000, E1   +58.900, E3 -261261.177}
SPL {X  -159.990, Y  +621.342, Z    +0.000, E1   +58.904, E3 -261270.685}
SPL {X  -159.990, Y  +629.920, Z    +0.000, E1   +58.912, E3 -261281.657}
SPL {X  -159.990, Y  +642.398, Z    +0.000, E1   +58.947, E3 -261297.565}
SPL {X  -159.990, Y  +654.206, Z    +0.000, E1   +58.908, E3 -261312.736}
SPL {X  -159.990, Y  +661.562, Z    +0.000, E1   +58.900, E3 -261322.164}
SPL {X  -159.990, Y  +670.328, Z    +0.000, E1   +58.911, E3 -261333.363}
SPL {X  -159.795, Y  +679.404, Z    +0.000, E1   +58.876, E3 -261345.188}
SPL {X  -159.282, Y  +686.534, Z    +0.000, E1   +58.787, E3 -261354.862}
SPL {X  -158.463, Y  +693.553, Z    +0.000, E1   +58.665, E3 -261364.703}
SPL {X  -157.294, Y  +700.745, Z    +0.000, E1   +58.469, E3 -261375.153}
SPL {X  -156.031, Y  +706.871, Z    +0.000, E1   +58.260, E3 -261384.299}
SPL {X  -154.558, Y  +712.835, Z    +0.000, E1   +58.028, E3 -261393.426}
SPL {X  -152.750, Y  +719.085, Z    +0.000, E1   +57.721, E3 -261403.272}
SPL {X  -150.741, Y  +725.111, Z    +0.000, E1   +57.387, E3 -261412.976}
SPL {X  -148.665, Y  +730.623, Z    +0.000, E1   +57.007, E3 -261422.125}
SPL {X  -146.664, Y  +735.425, Z    +0.000, E1   +56.657, E3 -261430.215}
SPL {X  -143.496, Y  +742.251, Z    +0.000, E1   +56.124, E3 -261441.908}
SPL {X  -140.752, Y  +747.564, Z    +0.000, E1   +55.554, E3 -261451.316}
SPL {X  -138.492, Y  +751.605, Z    +0.000, E1   +55.137, E3 -261458.507}
SPL {X  -124.324, Y  +772.199, Z    +0.000, E1   +48.708, E3 -261537.515}
ENDSPLINE

SPLINE
SPL {X  -129.118, Y  +765.975, Z    +0.000, E1   +43.713, E3 -261602.000}
SPL {X  -146.252, Y  +736.362, Z    +0.000, E1   +34.795, E3 -261651.178}
SPL {X  -155.916, Y  +707.374, Z    +0.000, E1   +22.878, E3 -261668.064}
SPL {X  -159.039, Y  +688.920, Z    +0.000, E1   +13.016, E3 -261673.298}
SPL {X  -159.777, Y  +679.762, Z    +0.000, E1    +7.372, E3 -261674.754}
SPL {X  -159.984, Y  +672.872, Z    +0.000, E1    +2.784, E3 -261675.350}
SPL {X  -159.990, Y  +668.898, Z    +0.000, E1    -0.346, E3 -261675.508}
SPL {X  -159.990, Y  +666.084, Z    +0.000, E1    -3.512, E3 -261675.631}
SPL {X  -159.990, Y  +662.904, Z    +0.000, E1    -7.618, E3 -261675.870}
SPL {X  -159.990, Y  +658.509, Z    +0.000, E1   -13.882, E3 -261676.406}
SPL {X  -159.990, Y  +652.317, Z    +0.000, E1   -22.778, E3 -261677.542}
SPL {X  -159.990, Y  +640.689, Z    +0.000, E1   -37.390, E3 -261679.084}
SPL {X  -159.990, Y  +585.634, Z    +0.000, E1   -68.681, E3 -261679.708}
SPL {X  -159.990, Y  +457.771, Z    +0.000, E1   -68.079, E3 -261770.270}
SPL {X  -159.990, Y  +453.218, Z    +0.000, E1   -67.322, E3 -261780.705}
SPL {X  -159.990, Y  +450.256, Z    +0.000, E1   -66.188, E3 -261792.638}
SPL {X  -159.990, Y  +445.667, Z    +0.000, E1   -65.356, E3 -261803.549}
SPL {X  -159.990, Y  +439.738, Z    +0.000, E1   -64.716, E3 -261814.362}
SPL {X  -159.990, Y  +433.217, Z    +0.000, E1   -63.756, E3 -261828.506}
SPL {X  -159.990, Y  +425.111, Z    +0.000, E1   -62.687, E3 -261845.047}
SPL {X  -159.990, Y  +418.218, Z    +0.000, E1   -61.769, E3 -261859.161}
SPL {X  -159.990, Y  +412.274, Z    +0.000, E1   -61.123, E3 -261870.565}
SPL {X  -159.990, Y  +408.631, Z    +0.000, E1   -60.233, E3 -261881.027}
SPL {X  -159.990, Y  +402.821, Z    +0.000, E1   -59.334, E3 -261894.555}
SPL {X  -159.990, Y  +395.849, Z    +0.000, E1   -58.799, E3 -261906.819}
SPL {X  -159.990, Y  +387.403, Z    +0.000, E1   -58.805, E3 -261917.665}
SPL {X  -159.948, Y  +378.844, Z    +0.000, E1   -58.798, E3 -261928.705}
SPL {X  -159.570, Y  +370.916, Z    +0.000, E1   -58.738, E3 -261939.300}
SPL {X  -158.865, Y  +363.563, Z    +0.000, E1   -58.615, E3 -261949.510}
SPL {X  -157.976, Y  +357.197, Z    +0.000, E1   -58.476, E3 -261958.611}
SPL {X  -156.730, Y  +350.368, Z    +0.000, E1   -58.276, E3 -261968.706}
SPL {X  -155.026, Y  +342.956, Z    +0.000, E1   -58.003, E3 -261979.978}
SPL {X  -152.946, Y  +335.551, Z    +0.000, E1   -57.653, E3 -261991.626}
SPL {X  -150.105, Y  +327.135, Z    +0.000, E1   -57.196, E3 -262005.246}
SPL {X  -146.578, Y  +318.377, Z    +0.000, E1   -56.572, E3 -262019.939}
SPL {X  -143.463, Y  +311.683, Z    +0.000, E1   -55.972, E3 -262031.552}
SPL {X  -140.858, Y  +306.633, Z    +0.000, E1   -55.477, E3 -262040.470}
SPL {X  -138.338, Y  +302.130, Z    +0.000, E1   -54.992, E3 -262048.519}
SPL {X  -124.427, Y  +281.929, Z    +0.000, E1   -46.852, E3 -262152.756}
ENDSPLINE

SPLINE
SPL {X  -148.251, Y  +322.346, Z    +0.000, E1   -33.039, E3 -262240.681}
SPL {X  -157.534, Y  +354.574, Z    +0.000, E1   -18.815, E3 -262257.510}
SPL {X  -159.548, Y  +370.614, Z    +0.000, E1    -9.656, E3 -262261.135}
SPL {X  -159.973, Y  +380.173, Z    +0.000, E1    -3.469, E3 -262262.202}
SPL {X  -159.990, Y  +384.078, Z    +0.000, E1    -0.490, E3 -262262.400}
SPL {X  -159.990, Y  +385.440, Z    +0.000, E1    +0.747, E3 -262262.441}
SPL {X  -159.990, Y  +388.179, Z    +0.000, E1    +3.660, E3 -262262.581}
SPL {X  -159.990, Y  +394.222, Z    +0.000, E1   +11.674, E3 -262263.175}
SPL {X  -159.990, Y  +403.976, Z    +0.000, E1   +25.456, E3 -262265.054}
SPL {X  -159.990, Y  +417.120, Z    +0.000, E1   +39.678, E3 -262269.086}
SPL {X  -159.990, Y  +456.927, Z    +0.000, E1   +55.382, E3 -262290.946}
SPL {X  -159.990, Y  +530.047, Z    +0.000, E1   +58.901, E3 -262360.780}
SPL {X  -159.990, Y  +538.035, Z    +0.000, E1   +58.900, E3 -262371.005}
SPL {X  -159.990, Y  +546.883, Z    +0.000, E1   +58.912, E3 -262382.309}
SPL {X  -159.990, Y  +555.949, Z    +0.000, E1   +58.900, E3 -262393.928}
SPL {X  -159.990, Y  +563.718, Z    +0.000, E1   +58.903, E3 -262403.848}
SPL {X  -159.990, Y  +571.529, Z    +0.000, E1   +58.906, E3 -262413.832}
SPL {X  -159.990, Y  +579.859, Z    +0.000, E1   +58.907, E3 -262424.492}
SPL {X  -159.990, Y  +588.526, Z    +0.000, E1   +58.910, E3 -262435.565}
SPL {X  -159.990, Y  +596.521, Z    +0.000, E1   +58.902, E3 -262445.824}
SPL {X  -159.990, Y  +605.444, Z    +0.000, E1   +58.918, E3 -262457.214}
SPL {X  -159.990, Y  +618.101, Z    +0.000, E1   +58.946, E3 -262473.361}
SPL {X  -159.990, Y  +629.920, Z    +0.000, E1   +58.912, E3 -262488.554}
SPL {X  -159.990, Y  +638.424, Z    +0.000, E1   +58.901, E3 -262499.454}
SPL {X  -159.990, Y  +645.995, Z    +0.000, E1   +58.900, E3 -262509.142}
SPL {X  -159.990, Y  +654.206, Z    +0.000, E1   +58.908, E3 -262519.632}
SPL {X  -159.990, Y  +661.562, Z    +0.000, E1   +58.900, E3 -262529.061}
SPL {X  -159.990, Y  +670.328, Z    +0.000, E1   +58.911, E3 -262540.260}
SPL {X  -159.795, Y  +679.404, Z    +0.000, E1   +58.876, E3 -262552.085}
SPL {X  -159.282, Y  +686.534, Z    +0.000, E1   +58.787, E3 -262561.759}
SPL {X  -158.463, Y  +693.553, Z    +0.000, E1   +58.665, E3 -262571.600}
SPL {X  -157.294, Y  +700.745, Z    +0.000, E1   +58.469, E3 -262582.050}
SPL {X  -156.031, Y  +706.871, Z    +0.000, E1   +58.260, E3 -262591.196}
SPL {X  -154.558, Y  +712.835, Z    +0.000, E1   +58.028, E3 -262600.323}
SPL {X  -152.750, Y  +719.085, Z    +0.000, E1   +57.721, E3 -262610.169}
SPL {X  -150.741, Y  +725.111, Z    +0.000, E1   +57.387, E3 -262619.873}
SPL {X  -148.665, Y  +730.623, Z    +0.000, E1   +57.007, E3 -262629.022}
SPL {X  -146.664, Y  +735.425, Z    +0.000, E1   +56.657, E3 -262637.112}
SPL {X  -143.496, Y  +742.251, Z    +0.000, E1   +56.124, E3 -262648.805}
SPL {X  -140.752, Y  +747.564, Z    +0.000, E1   +55.554, E3 -262658.212}
SPL {X  -138.492, Y  +751.605, Z    +0.000, E1   +55.137, E3 -262665.403}
SPL {X  -124.324, Y  +772.199, Z    +0.000, E1   +48.708, E3 -262744.411}
ENDSPLINE

SPLINE
SPL {X  -129.118, Y  +765.975, Z    +0.000, E1   +43.713, E3 -262808.897}
SPL {X  -146.252, Y  +736.362, Z    +0.000, E1   +34.795, E3 -262858.075}
SPL {X  -155.916, Y  +707.374, Z    +0.000, E1   +22.878, E3 -262874.960}
SPL {X  -159.039, Y  +688.920, Z    +0.000, E1   +13.016, E3 -262880.195}
SPL {X  -159.888, Y  +677.224, Z    +0.000, E1    +5.773, E3 -262881.907}
SPL {X  -159.990, Y  +671.755, Z    +0.000, E1    +1.905, E3 -262882.311}
SPL {X  -159.990, Y  +669.598, Z    +0.000, E1    +0.205, E3 -262882.384}
SPL {X  -159.990, Y  +667.097, Z    +0.000, E1    -2.190, E3 -262882.479}
SPL {X  -159.990, Y  +662.904, Z    +0.000, E1    -7.618, E3 -262882.767}
SPL {X  -159.990, Y  +658.509, Z    +0.000, E1   -13.882, E3 -262883.303}
SPL {X  -159.990, Y  +652.317, Z    +0.000, E1   -22.778, E3 -262884.438}
SPL {X  -159.990, Y  +640.689, Z    +0.000, E1   -37.390, E3 -262885.981}
SPL {X  -159.990, Y  +585.634, Z    +0.000, E1   -68.681, E3 -262886.605}
SPL {X  -159.990, Y  +457.771, Z    +0.000, E1   -68.079, E3 -262977.166}
SPL {X  -159.990, Y  +453.218, Z    +0.000, E1   -67.322, E3 -262987.601}
SPL {X  -159.990, Y  +450.256, Z    +0.000, E1   -66.188, E3 -262999.534}
SPL {X  -159.990, Y  +445.667, Z    +0.000, E1   -65.356, E3 -263010.446}
SPL {X  -159.990, Y  +439.738, Z    +0.000, E1   -64.716, E3 -263021.259}
SPL {X  -159.990, Y  +435.528, Z    +0.000, E1   -63.972, E3 -263031.134}
SPL {X  -159.990, Y  +429.021, Z    +0.000, E1   -63.228, E3 -263043.747}
SPL {X  -159.990, Y  +423.267, Z    +0.000, E1   -62.365, E3 -263056.045}
SPL {X  -159.990, Y  +418.218, Z    +0.000, E1   -61.769, E3 -263066.058}
SPL {X  -159.990, Y  +412.274, Z    +0.000, E1   -61.123, E3 -263077.462}
SPL {X  -159.990, Y  +408.631, Z    +0.000, E1   -60.233, E3 -263087.924}
SPL {X  -159.990, Y  +404.834, Z    +0.000, E1   -59.529, E3 -263097.379}
SPL {X  -159.990, Y  +397.866, Z    +0.000, E1   -58.924, E3 -263110.466}
SPL {X  -159.990, Y  +387.403, Z    +0.000, E1   -58.805, E3 -263124.562}
SPL {X  -159.948, Y  +378.844, Z    +0.000, E1   -58.798, E3 -263135.601}
SPL {X  -159.570, Y  +370.916, Z    +0.000, E1   -58.738, E3 -263146.197}
SPL {X  -158.865, Y  +363.563, Z    +0.000, E1   -58.615, E3 -263156.406}
SPL {X  -157.976, Y  +357.197, Z    +0.000, E1   -58.476, E3 -263165.507}
SPL {X  -156.730, Y  +350.368, Z    +0.000, E1   -58.276, E3 -263175.602}
SPL {X  -155.026, Y  +342.956, Z    +0.000, E1   -58.003, E3 -263186.875}
SPL {X  -152.946, Y  +335.551, Z    +0.000, E1   -57.653, E3 -263198.522}
SPL {X  -150.105, Y  +327.135, Z    +0.000, E1   -57.196, E3 -263212.143}
SPL {X  -146.578, Y  +318.377, Z    +0.000, E1   -56.572, E3 -263226.835}
SPL {X  -143.463, Y  +311.683, Z    +0.000, E1   -55.972, E3 -263238.449}
SPL {X  -140.858, Y  +306.633, Z    +0.000, E1   -55.477, E3 -263247.366}
SPL {X  -138.338, Y  +302.130, Z    +0.000, E1   -54.992, E3 -263255.416}
SPL {X  -124.427, Y  +281.929, Z    +0.000, E1   -46.852, E3 -263359.652}
ENDSPLINE

SPLINE
SPL {X  -148.251, Y  +322.346, Z    +0.000, E1   -33.039, E3 -263447.577}
SPL {X  -157.534, Y  +354.574, Z    +0.000, E1   -18.815, E3 -263464.406}
SPL {X  -159.548, Y  +370.614, Z    +0.000, E1    -9.656, E3 -263468.032}
SPL {X  -159.928, Y  +378.035, Z    +0.000, E1    -4.866, E3 -263468.947}
SPL {X  -159.990, Y  +383.381, Z    +0.000, E1    -1.123, E3 -263469.268}
SPL {X  -159.990, Y  +386.348, Z    +0.000, E1    +1.571, E3 -263469.377}
SPL {X  -159.990, Y  +391.422, Z    +0.000, E1    +7.757, E3 -263469.751}
SPL {X  -159.990, Y  +399.099, Z    +0.000, E1   +18.787, E3 -263470.858}
SPL {X  -159.990, Y  +406.316, Z    +0.000, E1   +28.569, E3 -263472.535}
SPL {X  -159.990, Y  +417.120, Z    +0.000, E1   +39.678, E3 -263475.982}
SPL {X  -159.990, Y  +456.927, Z    +0.000, E1   +55.382, E3 -263497.842}
SPL {X  -159.990, Y  +530.047, Z    +0.000, E1   +58.901, E3 -263567.676}
SPL {X  -159.990, Y  +538.035, Z    +0.000, E1   +58.900, E3 -263577.902}
SPL {X  -159.990, Y  +546.883, Z    +0.000, E1   +58.912, E3 -263589.205}
SPL {X  -159.990, Y  +555.949, Z    +0.000, E1   +58.900, E3 -263600.825}
SPL {X  -159.990, Y  +563.718, Z    +0.000, E1   +58.903, E3 -263610.745}
SPL {X  -159.990, Y  +571.529, Z    +0.000, E1   +58.906, E3 -263620.729}
SPL {X  -159.990, Y  +579.859, Z    +0.000, E1   +58.907, E3 -263631.388}
SPL {X  -159.990, Y  +588.526, Z    +0.000, E1   +58.910, E3 -263642.462}
SPL {X  -159.990, Y  +596.521, Z    +0.000, E1   +58.902, E3 -263652.721}
SPL {X  -159.990, Y  +605.444, Z    +0.000, E1   +58.918, E3 -263664.110}
SPL {X  -159.990, Y  +618.101, Z    +0.000, E1   +58.946, E3 -263680.257}
SPL {X  -159.990, Y  +629.920, Z    +0.000, E1   +58.912, E3 -263695.450}
SPL {X  -159.990, Y  +638.424, Z    +0.000, E1   +58.901, E3 -263706.350}
SPL {X  -159.990, Y  +645.995, Z    +0.000, E1   +58.900, E3 -263716.038}
SPL {X  -159.990, Y  +654.206, Z    +0.000, E1   +58.908, E3 -263726.529}
SPL {X  -159.990, Y  +661.562, Z    +0.000, E1   +58.900, E3 -263735.957}
SPL {X  -159.990, Y  +670.328, Z    +0.000, E1   +58.911, E3 -263747.156}
SPL {X  -159.795, Y  +679.404, Z    +0.000, E1   +58.876, E3 -263758.982}
SPL {X  -159.282, Y  +686.534, Z    +0.000, E1   +58.787, E3 -263768.655}
SPL {X  -158.463, Y  +693.553, Z    +0.000, E1   +58.665, E3 -263778.496}
SPL {X  -157.294, Y  +700.745, Z    +0.000, E1   +58.469, E3 -263788.946}
SPL {X  -156.031, Y  +706.871, Z    +0.000, E1   +58.260, E3 -263798.092}
SPL {X  -154.558, Y  +712.835, Z    +0.000, E1   +58.028, E3 -263807.219}
SPL {X  -152.750, Y  +719.085, Z    +0.000, E1   +57.721, E3 -263817.065}
SPL {X  -150.741, Y  +725.111, Z    +0.000, E1   +57.387, E3 -263826.769}
SPL {X  -148.665, Y  +730.623, Z    +0.000, E1   +57.007, E3 -263835.918}
SPL {X  -146.664, Y  +735.425, Z    +0.000, E1   +56.657, E3 -263844.008}
SPL {X  -143.496, Y  +742.251, Z    +0.000, E1   +56.124, E3 -263855.701}
SPL {X  -140.752, Y  +747.564, Z    +0.000, E1   +55.554, E3 -263865.109}
SPL {X  -138.492, Y  +751.605, Z    +0.000, E1   +55.137, E3 -263872.300}
SPL {X  -124.324, Y  +772.199, Z    +0.000, E1   +48.708, E3 -263951.308}
ENDSPLINE

SPLINE
SPL {X  -129.118, Y  +765.975, Z    +0.000, E1   +43.713, E3 -264015.793}
SPL {X  -146.252, Y  +736.362, Z    +0.000, E1   +34.795, E3 -264064.971}
SPL {X  -154.088, Y  +714.555, Z    +0.000, E1   +26.177, E3 -264078.987}
SPL {X  -156.688, Y  +703.837, Z    +0.000, E1   +21.096, E3 -264083.159}
SPL {X  -159.039, Y  +688.920, Z    +0.000, E1   +13.016, E3 -264087.091}
SPL {X  -159.888, Y  +677.224, Z    +0.000, E1    +5.773, E3 -264088.804}
SPL {X  -159.990, Y  +670.275, Z    +0.000, E1    +0.854, E3 -264089.258}
SPL {X  -159.990, Y  +667.097, Z    +0.000, E1    -2.190, E3 -264089.375}
SPL {X  -159.990, Y  +662.904, Z    +0.000, E1    -7.618, E3 -264089.663}
SPL {X  -159.990, Y  +658.509, Z    +0.000, E1   -13.882, E3 -264090.199}
SPL {X  -159.990, Y  +652.317, Z    +0.000, E1   -22.778, E3 -264091.335}
SPL {X  -159.990, Y  +640.689, Z    +0.000, E1   -37.390, E3 -264092.877}
SPL {X  -159.990, Y  +585.634, Z    +0.000, E1   -68.681, E3 -264093.501}
SPL {X  -159.990, Y  +457.771, Z    +0.000, E1   -68.079, E3 -264184.063}
SPL {X  -159.990, Y  +453.218, Z    +0.000, E1   -67.322, E3 -264194.498}
SPL {X  -159.990, Y  +450.256, Z    +0.000, E1   -66.188, E3 -264206.431}
SPL {X  -159.990, Y  +445.667, Z    +0.000, E1   -65.356, E3 -264217.342}
SPL {X  -159.990, Y  +439.738, Z    +0.000, E1   -64.716, E3 -264228.155}
SPL {X  -159.990, Y  +435.528, Z    +0.000, E1   -63.972, E3 -264238.031}
SPL {X  -159.990, Y  +429.021, Z    +0.000, E1   -63.228, E3 -264250.644}
SPL {X  -159.990, Y  +423.267, Z    +0.000, E1   -62.365, E3 -264262.942}
SPL {X  -159.990, Y  +418.218, Z    +0.000, E1   -61.769, E3 -264272.954}
SPL {X  -159.990, Y  +412.274, Z    +0.000, E1   -61.123, E3 -264284.358}
SPL {X  -159.990, Y  +408.631, Z    +0.000, E1   -60.233, E3 -264294.821}
SPL {X  -159.990, Y  +404.834, Z    +0.000, E1   -59.529, E3 -264304.276}
SPL {X  -159.990, Y  +397.866, Z    +0.000, E1   -58.924, E3 -264317.363}
SPL {X  -159.990, Y  +387.403, Z    +0.000, E1   -58.805, E3 -264331.458}
SPL {X  -159.948, Y  +378.844, Z    +0.000, E1   -58.798, E3 -264342.498}
SPL {X  -159.570, Y  +370.916, Z    +0.000, E1   -58.738, E3 -264353.093}
SPL {X  -158.865, Y  +363.563, Z    +0.000, E1   -58.615, E3 -264363.303}
SPL {X  -157.976, Y  +357.197, Z    +0.000, E1   -58.476, E3 -264372.404}
SPL {X  -156.730, Y  +350.368, Z    +0.000, E1   -58.276, E3 -264382.499}
SPL {X  -155.026, Y  +342.956, Z    +0.000, E1   -58.003, E3 -264393.771}
SPL {X  -152.946, Y  +335.551, Z    +0.000, E1   -57.653, E3 -264405.419}
SPL {X  -150.899, Y  +329.336, Z    +0.000, E1   -57.290, E3 -264415.485}
SPL {X  -149.179, Y  +324.687, Z    +0.000, E1   -56.983, E3 -264423.174}
SPL {X  -146.578, Y  +318.377, Z    +0.000, E1   -56.572, E3 -264433.732}
SPL {X  -143.463, Y  +311.683, Z    +0.000, E1   -55.972, E3 -264445.346}
SPL {X  -140.858, Y  +306.633, Z    +0.000, E1   -55.477, E3 -264454.263}
SPL {X  -138.338, Y  +302.130, Z    +0.000, E1   -54.992, E3 -264462.312}
SPL {X  -124.427, Y  +281.929, Z    +0.000, E1   -46.852, E3 -264566.549}
ENDSPLINE

SPLINE
SPL {X  -138.506, Y  +302.419, Z    +0.000, E1   -39.451, E3 -264632.523}
SPL {X  -149.686, Y  +326.013, Z    +0.000, E1   -31.658, E3 -264657.660}
SPL {X  -156.481, Y  +349.177, Z    +0.000, E1   -21.514, E3 -264669.657}
SPL {X  -159.327, Y  +367.953, Z    +0.000, E1   -11.342, E3 -264674.448}
SPL {X  -159.973, Y  +380.173, Z    +0.000, E1    -3.469, E3 -264675.995}
SPL {X  -159.990, Y  +384.078, Z    +0.000, E1    -0.490, E3 -264676.193}
SPL {X  -159.990, Y  +385.440, Z    +0.000, E1    +0.747, E3 -264676.234}
SPL {X  -159.990, Y  +388.179, Z    +0.000, E1    +3.660, E3 -264676.374}
SPL {X  -159.990, Y  +394.222, Z    +0.000, E1   +11.674, E3 -264676.968}
SPL {X  -159.990, Y  +403.976, Z    +0.000, E1   +25.456, E3 -264678.847}
SPL {X  -159.990, Y  +417.120, Z    +0.000, E1   +39.678, E3 -264682.879}
SPL {X  -159.990, Y  +456.927, Z    +0.000, E1   +55.382, E3 -264704.739}
SPL {X  -159.990, Y  +530.047, Z    +0.000, E1   +58.901, E3 -264774.573}
SPL {X  -159.990, Y  +538.035, Z    +0.000, E1   +58.900, E3 -264784.798}
SPL {X  -159.990, Y  +546.883, Z    +0.000, E1   +58.912, E3 -264796.102}
SPL {X  -159.990, Y  +555.949, Z    +0.000, E1   +58.900, E3 -264807.721}
SPL {X  -159.990, Y  +563.718, Z    +0.000, E1   +58.903, E3 -264817.641}
SPL {X  -159.990, Y  +571.529, Z    +0.000, E1   +58.906, E3 -264827.626}
SPL {X  -159.990, Y  +579.859, Z    +0.000, E1   +58.907, E3 -264838.285}
SPL {X  -159.990, Y  +588.526, Z    +0.000, E1   +58.910, E3 -264849.358}
SPL {X  -159.990, Y  +596.521, Z    +0.000, E1   +58.902, E3 -264859.618}
SPL {X  -159.990, Y  +605.444, Z    +0.000, E1   +58.918, E3 -264871.007}
SPL {X  -159.990, Y  +613.908, Z    +0.000, E1   +58.900, E3 -264881.866}
SPL {X  -159.990, Y  +621.342, Z    +0.000, E1   +58.904, E3 -264891.374}
SPL {X  -159.990, Y  +629.920, Z    +0.000, E1   +58.912, E3 -264902.347}
SPL {X  -159.990, Y  +642.398, Z    +0.000, E1   +58.947, E3 -264918.254}
SPL {X  -159.990, Y  +654.206, Z    +0.000, E1   +58.908, E3 -264933.425}
SPL {X  -159.990, Y  +661.562, Z    +0.000, E1   +58.900, E3 -264942.854}
SPL {X  -159.990, Y  +670.328, Z    +0.000, E1   +58.911, E3 -264954.053}
SPL {X  -159.795, Y  +679.404, Z    +0.000, E1   +58.876, E3 -264965.878}
SPL {X  -159.282, Y  +686.534, Z    +0.000, E1   +58.787, E3 -264975.552}
SPL {X  -158.463, Y  +693.553, Z    +0.000, E1   +58.665, E3 -264985.393}
SPL {X  -157.294, Y  +700.745, Z    +0.000, E1   +58.469, E3 -264995.843}
SPL {X  -156.031, Y  +706.871, Z    +0.000, E1   +58.260, E3 -265004.989}
SPL {X  -154.558, Y  +712.835, Z    +0.000, E1   +58.028, E3 -265014.116}
SPL {X  -152.750, Y  +719.085, Z    +0.000, E1   +57.721, E3 -265023.962}
SPL {X  -150.741, Y  +725.111, Z    +0.000, E1   +57.387, E3 -265033.666}
SPL {X  -148.665, Y  +730.623, Z    +0.000, E1   +57.007, E3 -265042.815}
SPL {X  -146.664, Y  +735.425, Z    +0.000, E1   +56.657, E3 -265050.905}
SPL {X  -143.496, Y  +742.251, Z    +0.000, E1   +56.124, E3 -265062.598}
SPL {X  -140.752, Y  +747.564, Z    +0.000, E1   +55.554, E3 -265072.005}
SPL {X  -138.492, Y  +751.605, Z    +0.000, E1   +55.137, E3 -265079.196}
SPL {X  -124.324, Y  +772.199, Z    +0.000, E1   +48.708, E3 -265158.205}
ENDSPLINE

SPLINE
SPL {X  -129.118, Y  +765.975, Z    +0.000, E1   +43.713, E3 -265222.690}
SPL {X  -146.252, Y  +736.362, Z    +0.000, E1   +34.795, E3 -265271.868}
SPL {X  -154.088, Y  +714.555, Z    +0.000, E1   +26.177, E3 -265285.884}
SPL {X  -156.688, Y  +703.837, Z    +0.000, E1   +21.096, E3 -265290.056}
SPL {X  -159.039, Y  +688.920, Z    +0.000, E1   +13.016, E3 -265293.988}
SPL {X  -159.888, Y  +677.224, Z    +0.000, E1    +5.773, E3 -265295.701}
SPL {X  -159.990, Y  +671.755, Z    +0.000, E1    +1.905, E3 -265296.104}
SPL {X  -159.990, Y  +669.598, Z    +0.000, E1    +0.205, E3 -265296.177}
SPL {X  -159.990, Y  +667.097, Z    +0.000, E1    -2.190, E3 -265296.272}
SPL {X  -159.990, Y  +662.904, Z    +0.000, E1    -7.618, E3 -265296.560}
SPL {X  -159.990, Y  +658.509, Z    +0.000, E1   -13.882, E3 -265297.096}
SPL {X  -159.990, Y  +652.317, Z    +0.000, E1   -22.778, E3 -265298.231}
SPL {X  -159.990, Y  +641.893, Z    +0.000, E1   -35.310, E3 -265301.196}
SPL {X  -159.990, Y  +636.123, Z    +0.000, E1   -46.139, E3 -265294.261}
SPL {X  -159.990, Y  +585.634, Z    +0.000, E1   -68.681, E3 -265300.398}
SPL {X  -159.990, Y  +457.771, Z    +0.000, E1   -68.079, E3 -265390.959}
SPL {X  -159.990, Y  +453.218, Z    +0.000, E1   -67.322, E3 -265401.395}
SPL {X  -159.990, Y  +450.256, Z    +0.000, E1   -66.188, E3 -265413.327}
SPL {X  -159.990, Y  +445.667, Z    +0.000, E1   -65.356, E3 -265424.239}
SPL {X  -159.990, Y  +439.738, Z    +0.000, E1   -64.716, E3 -265435.052}
SPL {X  -159.990, Y  +435.528, Z    +0.000, E1   -63.972, E3 -265444.927}
SPL {X  -159.990, Y  +429.021, Z    +0.000, E1   -63.228, E3 -265457.540}
SPL {X  -159.990, Y  +423.267, Z    +0.000, E1   -62.365, E3 -265469.838}
SPL {X  -159.990, Y  +418.218, Z    +0.000, E1   -61.769, E3 -265479.851}
SPL {X  -159.990, Y  +412.274, Z    +0.000, E1   -61.123, E3 -265491.255}
SPL {X  -159.990, Y  +408.631, Z    +0.000, E1   -60.233, E3 -265501.717}
SPL {X  -159.990, Y  +404.834, Z    +0.000, E1   -59.529, E3 -265511.172}
SPL {X  -159.990, Y  +397.866, Z    +0.000, E1   -58.924, E3 -265524.259}
SPL {X  -159.990, Y  +387.403, Z    +0.000, E1   -58.805, E3 -265538.355}
SPL {X  -159.948, Y  +378.844, Z    +0.000, E1   -58.798, E3 -265549.394}
SPL {X  -159.570, Y  +370.916, Z    +0.000, E1   -58.738, E3 -265559.990}
SPL {X  -158.865, Y  +363.563, Z    +0.000, E1   -58.615, E3 -265570.199}
SPL {X  -157.976, Y  +357.197, Z    +0.000, E1   -58.476, E3 -265579.300}
SPL {X  -156.730, Y  +350.368, Z    +0.000, E1   -58.276, E3 -265589.395}
SPL {X  -155.026, Y  +342.956, Z    +0.000, E1   -58.003, E3 -265600.668}
SPL {X  -152.946, Y  +335.551, Z    +0.000, E1   -57.653, E3 -265612.315}
SPL {X  -150.899, Y  +329.336, Z    +0.000, E1   -57.290, E3 -265622.381}
SPL {X  -149.179, Y  +324.687, Z    +0.000, E1   -56.983, E3 -265630.071}
SPL {X  -147.281, Y  +320.009, Z    +0.000, E1   -56.662, E3 -265637.897}
SPL {X  -144.114, Y  +313.017, Z    +0.000, E1   -56.131, E3 -265649.864}
SPL {X  -140.858, Y  +306.633, Z    +0.000, E1   -55.477, E3 -265661.159}
SPL {X  -138.338, Y  +302.130, Z    +0.000, E1   -54.992, E3 -265669.209}
SPL {X  -124.427, Y  +281.929, Z    +0.000, E1   -46.852, E3 -265773.445}
ENDSPLINE

SPLINE
SPL {X  -148.251, Y  +322.346, Z    +0.000, E1   -33.039, E3 -265861.370}
SPL {X  -157.534, Y  +354.574, Z    +0.000, E1   -18.815, E3 -265878.199}
SPL {X  -159.548, Y  +370.614, Z    +0.000, E1    -9.656, E3 -265881.825}
SPL {X  -159.973, Y  +380.173, Z    +0.000, E1    -3.469, E3 -265882.892}
SPL {X  -159.990, Y  +384.078, Z    +0.000, E1    -0.490, E3 -265883.089}
SPL {X  -159.990, Y  +386.348, Z    +0.000, E1    +1.571, E3 -265883.170}
SPL {X  -159.990, Y  +391.422, Z    +0.000, E1    +7.757, E3 -265883.544}
SPL {X  -159.990, Y  +399.099, Z    +0.000, E1   +18.787, E3 -265884.651}
SPL {X  -159.990, Y  +406.316, Z    +0.000, E1   +28.569, E3 -265886.328}
SPL {X  -159.990, Y  +417.120, Z    +0.000, E1   +39.678, E3 -265889.775}
SPL {X  -159.990, Y  +456.927, Z    +0.000, E1   +55.382, E3 -265911.635}
SPL {X  -159.990, Y  +530.047, Z    +0.000, E1   +58.901, E3 -265981.469}
SPL {X  -159.990, Y  +538.035, Z    +0.000, E1   +58.900, E3 -265991.695}
SPL {X  -159.990, Y  +546.883, Z    +0.000, E1   +58.912, E3 -266002.998}
SPL {X  -159.990, Y  +555.949, Z    +0.000, E1   +58.900, E3 -266014.618}
SPL {X  -159.990, Y  +563.718, Z    +0.000, E1   +58.903, E3 -266024.538}
SPL {X  -159.990, Y  +571.529, Z    +0.000, E1   +58.906, E3 -266034.522}
SPL {X  -159.990, Y  +579.859, Z    +0.000, E1   +58.907, E3 -266045.181}
SPL {X  -159.990, Y  +588.526, Z    +0.000, E1   +58.910, E3 -266056.255}
SPL {X  -159.990, Y  +596.521, Z    +0.000, E1   +58.902, E3 -266066.514}
SPL {X  -159.990, Y  +605.444, Z    +0.000, E1   +58.918, E3 -266077.904}
SPL {X  -159.990, Y  +613.908, Z    +0.000, E1   +58.900, E3 -266088.763}
SPL {X  -159.990, Y  +621.342, Z    +0.000, E1   +58.904, E3 -266098.271}
SPL {X  -159.990, Y  +629.920, Z    +0.000, E1   +58.912, E3 -266109.243}
SPL {X  -159.990, Y  +642.398, Z    +0.000, E1   +58.947, E3 -266125.151}
SPL {X  -159.990, Y  +654.206, Z    +0.000, E1   +58.908, E3 -266140.322}
SPL {X  -159.990, Y  +661.562, Z    +0.000, E1   +58.900, E3 -266149.750}
SPL {X  -159.990, Y  +670.328, Z    +0.000, E1   +58.911, E3 -266160.949}
SPL {X  -159.795, Y  +679.404, Z    +0.000, E1   +58.876, E3 -266172.775}
SPL {X  -159.282, Y  +686.534, Z    +0.000, E1   +58.787, E3 -266182.448}
SPL {X  -158.463, Y  +693.553, Z    +0.000, E1   +58.665, E3 -266192.289}
SPL {X  -157.294, Y  +700.745, Z    +0.000, E1   +58.469, E3 -266202.740}
SPL {X  -156.031, Y  +706.871, Z    +0.000, E1   +58.260, E3 -266211.885}
SPL {X  -154.558, Y  +712.835, Z    +0.000, E1   +58.028, E3 -266221.012}
SPL {X  -152.750, Y  +719.085, Z    +0.000, E1   +57.721, E3 -266230.859}
SPL {X  -150.741, Y  +725.111, Z    +0.000, E1   +57.387, E3 -266240.563}
SPL {X  -148.665, Y  +730.623, Z    +0.000, E1   +57.007, E3 -266249.711}
SPL {X  -146.664, Y  +735.425, Z    +0.000, E1   +56.657, E3 -266257.801}
SPL {X  -144.631, Y  +739.900, Z    +0.000, E1   +56.280, E3 -266265.487}
SPL {X  -141.795, Y  +745.600, Z    +0.000, E1   +55.801, E3 -266275.370}
SPL {X  -138.492, Y  +751.605, Z    +0.000, E1   +55.137, E3 -266286.093}
SPL {X  -124.324, Y  +772.199, Z    +0.000, E1   +48.708, E3 -266365.101}
ENDSPLINE

SPLINE
SPL {X  -129.118, Y  +765.975, Z    +0.000, E1   +43.713, E3 -266429.587}
SPL {X  -146.252, Y  +736.362, Z    +0.000, E1   +34.795, E3 -266478.764}
SPL {X  -154.088, Y  +714.555, Z    +0.000, E1   +26.177, E3 -266492.781}
SPL {X  -156.688, Y  +703.837, Z    +0.000, E1   +21.096, E3 -266496.952}
SPL {X  -159.039, Y  +688.920, Z    +0.000, E1   +13.016, E3 -266500.884}
SPL {X  -159.888, Y  +677.224, Z    +0.000, E1    +5.773, E3 -266502.597}
SPL {X  -159.990, Y  +670.275, Z    +0.000, E1    +0.854, E3 -266503.051}
SPL {X  -159.990, Y  +667.097, Z    +0.000, E1    -2.190, E3 -266503.168}
SPL {X  -159.990, Y  +662.904, Z    +0.000, E1    -7.618, E3 -266503.457}
SPL {X  -159.990, Y  +658.509, Z    +0.000, E1   -13.882, E3 -266503.992}
SPL {X  -159.990, Y  +652.317, Z    +0.000, E1   -22.778, E3 -266505.128}
SPL {X  -159.990, Y  +640.689, Z    +0.000, E1   -37.390, E3 -266506.670}
SPL {X  -159.990, Y  +585.634, Z    +0.000, E1   -68.681, E3 -266507.295}
SPL {X  -159.990, Y  +457.771, Z    +0.000, E1   -68.079, E3 -266597.856}
SPL {X  -159.990, Y  +453.218, Z    +0.000, E1   -67.322, E3 -266608.291}
SPL {X  -159.990, Y  +450.256, Z    +0.000, E1   -66.188, E3 -266620.224}
SPL {X  -159.990, Y  +445.667, Z    +0.000, E1   -65.356, E3 -266631.136}
SPL {X  -159.990, Y  +439.738, Z    +0.000, E1   -64.716, E3 -266641.948}
SPL {X  -159.990, Y  +435.528, Z    +0.000, E1   -63.972, E3 -266651.824}
SPL {X  -159.990, Y  +429.021, Z    +0.000, E1   -63.228, E3 -266664.437}
SPL {X  -159.990, Y  +423.267, Z    +0.000, E1   -62.365, E3 -266676.735}
SPL {X  -159.990, Y  +418.218, Z    +0.000, E1   -61.769, E3 -266686.747}
SPL {X  -159.990, Y  +412.274, Z    +0.000, E1   -61.123, E3 -266698.151}
SPL {X  -159.990, Y  +408.631, Z    +0.000, E1   -60.233, E3 -266708.614}
SPL {X  -159.990, Y  +402.720, Z    +0.000, E1   -59.334, E3 -266722.274}
ENDSPLINE

SPLINE
SPL {X  -159.990, Y  +412.718, Z    +0.000, E1   -54.930, E3 -266737.032}
ENDSPLINE

SPLINE
SPL {X  -159.990, Y  +405.235, Z    +0.000, E1   -54.902, E3 -266748.245}
SPL {X  -159.990, Y  +400.284, Z    +0.000, E1   -54.897, E3 -266755.640}
SPL {X  -159.990, Y  +391.119, Z    +0.000, E1   -54.948, E3 -266769.228}
SPL {X  -159.951, Y  +378.972, Z    +0.000, E1   -54.929, E3 -266787.406}
SPL {X  -159.499, Y  +369.977, Z    +0.000, E1   -54.827, E3 -266801.319}
SPL {X  -158.803, Y  +363.045, Z    +0.000, E1   -54.709, E3 -266812.387}
SPL {X  -157.732, Y  +355.717, Z    +0.000, E1   -54.540, E3 -266824.410}
SPL {X  -156.235, Y  +348.039, Z    +0.000, E1   -54.281, E3 -266837.421}
SPL {X  -154.716, Y  +341.761, Z    +0.000, E1   -53.995, E3 -266848.378}
SPL {X  -152.882, Y  +335.340, Z    +0.000, E1   -53.695, E3 -266859.780}
SPL {X  -151.019, Y  +329.680, Z    +0.000, E1   -53.334, E3 -266870.137}
SPL {X  -148.682, Y  +323.421, Z    +0.000, E1   -52.939, E3 -266881.739}
SPL {X  -145.914, Y  +316.881, Z    +0.000, E1   -52.402, E3 -266894.203}
SPL {X  -142.795, Y  +310.344, Z    +0.000, E1   -51.829, E3 -266906.859}
SPL {X  -132.354, Y  +292.616, Z    +0.000, E1   -44.164, E3 -267005.271}
ENDSPLINE

SPLINE
SPL {X  -150.910, Y  +329.369, Z    +0.000, E1   -29.678, E3 -267077.667}
SPL {X  -156.829, Y  +350.854, Z    +0.000, E1   -20.141, E3 -267090.219}
SPL {X  -159.049, Y  +365.169, Z    +0.000, E1   -12.580, E3 -267094.963}
SPL {X  -159.776, Y  +374.231, Z    +0.000, E1    -7.281, E3 -267096.850}
SPL {X  -159.986, Y  +381.380, Z    +0.000, E1    -2.685, E3 -267097.696}
SPL {X  -159.990, Y  +384.493, Z    +0.000, E1    -0.324, E3 -267097.904}
SPL {X  -159.990, Y  +387.327, Z    +0.000, E1    +2.137, E3 -267098.086}
SPL {X  -159.990, Y  +390.622, Z    +0.000, E1    +5.876, E3 -267098.380}
SPL {X  -159.990, Y  +394.493, Z    +0.000, E1   +10.512, E3 -267098.903}
SPL {X  -159.990, Y  +401.377, Z    +0.000, E1   +19.398, E3 -267100.357}
SPL {X  -159.990, Y  +411.365, Z    +0.000, E1   +30.630, E3 -267103.566}
SPL {X  -159.990, Y  +450.467, Z    +0.000, E1   +50.183, E3 -267127.214}
SPL {X  -159.990, Y  +509.934, Z    +0.000, E1   +54.923, E3 -267189.833}
SPL {X  -159.990, Y  +516.848, Z    +0.000, E1   +54.930, E3 -267200.121}
SPL {X  -159.990, Y  +524.818, Z    +0.000, E1   +54.933, E3 -267211.993}
SPL {X  -159.990, Y  +532.100, Z    +0.000, E1   +54.924, E3 -267222.846}
SPL {X  -159.990, Y  +539.391, Z    +0.000, E1   +54.933, E3 -267233.698}
SPL {X  -159.990, Y  +546.283, Z    +0.000, E1   +54.924, E3 -267243.970}
SPL {X  -159.990, Y  +553.734, Z    +0.000, E1   +54.938, E3 -267255.057}
SPL {X  -159.990, Y  +564.956, Z    +0.000, E1   +54.973, E3 -267271.728}
SPL {X  -159.990, Y  +575.140, Z    +0.000, E1   +54.928, E3 -267286.961}
SPL {X  -159.990, Y  +581.046, Z    +0.000, E1   +54.920, E3 -267295.774}
SPL {X  -159.990, Y  +588.063, Z    +0.000, E1   +54.931, E3 -267306.209}
SPL {X  -159.990, Y  +595.273, Z    +0.000, E1   +54.928, E3 -267316.932}
SPL {X  -159.990, Y  +602.326, Z    +0.000, E1   +54.932, E3 -267327.432}
SPL {X  -159.990, Y  +610.296, Z    +0.000, E1   +54.937, E3 -267339.302}
SPL {X  -159.990, Y  +618.534, Z    +0.000, E1   +54.942, E3 -267351.539}
SPL {X  -159.990, Y  +625.928, Z    +0.000, E1   +54.931, E3 -267362.564}
SPL {X  -159.990, Y  +633.423, Z    +0.000, E1   +54.943, E3 -267373.706}
SPL {X  -159.990, Y  +640.333, Z    +0.000, E1   +54.927, E3 -267384.020}
SPL {X  -159.990, Y  +648.272, Z    +0.000, E1   +54.961, E3 -267395.768}
SPL {X  -159.990, Y  +655.990, Z    +0.000, E1   +54.930, E3 -267407.315}
SPL {X  -159.990, Y  +665.734, Z    +0.000, E1   +54.984, E3 -267421.767}
SPL {X  -159.953, Y  +674.920, Z    +0.000, E1   +54.918, E3 -267435.578}
SPL {X  -159.714, Y  +680.893, Z    +0.000, E1   +54.890, E3 -267444.718}
SPL {X  -159.222, Y  +687.156, Z    +0.000, E1   +54.792, E3 -267454.606}
SPL {X  -158.388, Y  +694.082, Z    +0.000, E1   +54.679, E3 -267465.743}
SPL {X  -157.277, Y  +700.838, Z    +0.000, E1   +54.465, E3 -267477.000}
SPL {X  -156.153, Y  +706.327, Z    +0.000, E1   +54.274, E3 -267486.337}
SPL {X  -154.505, Y  +713.032, Z    +0.000, E1   +54.006, E3 -267497.998}
SPL {X  -152.808, Y  +718.896, Z    +0.000, E1   +53.679, E3 -267508.495}
SPL {X  -150.773, Y  +725.019, Z    +0.000, E1   +53.343, E3 -267519.627}
SPL {X  -148.029, Y  +732.198, Z    +0.000, E1   +52.831, E3 -267533.064}
SPL {X  -145.158, Y  +738.775, Z    +0.000, E1   +52.288, E3 -267545.649}
SPL {X  -142.385, Y  +744.461, Z    +0.000, E1   +51.729, E3 -267556.761}
SPL {X  -132.301, Y  +761.463, Z    +0.000, E1   +45.510, E3 -267634.500}
ENDSPLINE

